# B&R Automation Studio project AP124 (part 2)

#### Variables.var - Local variables
```iecst
VAR
	closeArms : BOOL; (*VISU:1..command to close the arms, 0...open arms*)
	cmdDown : BOOL; (*VISU: button to go with magazine down*)
	cmdUp : BOOL; (*VISU: go with magazine down*)
	diActivateMagazineSafetyCircuits : BOOL; (*magazine:3 funkce v 1 (reset safety+ovladaci obvody + start automatu pokud jede paletizace)*)
	diLeftArmClosed : BOOL; (*left arm is closed*)
	diLeftArmOpened : BOOL; (*left arm is opened*)
	diMagazineLooseChain : BOOL; (*lower HW end switch*)
	diMagazineLowerPosition : BOOL; (*magazine in lower position*)
	diMagazineMiddlePositon : BOOL; (*magazine in middle position*)
	diMagazineUpperHwEnd : BOOL; (*upper HW end switch*)
	diMagazineUpperPosition : BOOL; (*magazine in upper position*)
	diMotorProtectionP11 : BOOL; (*contactor for vertical movement, 1=OK*)
	diPalletOnConveyorP12 : BOOL; (*pallet detected on conveyor P12*)
	diRightArmClosed : BOOL; (*right arm is closed*)
	diRightArmOpened : BOOL; (*right arm is opened*)
	doCloseArms : BOOL; (*valve to close the arms*)
	doLedP11 : BOOL;
	doMagazineBrake : BOOL; (*1=brake released*)
	doMagazineDown : BOOL; (*contactor to go down*)
	doMagazineUp : BOOL; (*contactor to go up*)
	doOpenArms : BOOL; (*valve to open the arms*)
	lightCurtainP11 : BOOL; (*status of light curtain P11*)
	MTBasicsPWM_0 : MTBasicsPWM;
	readyToStart : BOOL;
	stateArms : StateArms; (*VISU:arms state*)
	stateAuto : StateAuto;
	stateMagazine : StateMagazine; (*VISU: current state of magazine*)
	TON_LeftRequest : TON;
	TON_RightRequest : TON;
	TON_VerticalMovement : TON;
	TP_Start : TP;
	TON_PalletOnConveyorP12 : TON;
	modeZoneMagazineOld : ModeZone;
END_VAR
```

#### horizontalArmsControl.st
```iecst
(* control of arms *)

ACTION HorizontalArmsControl:

	IF modeZoneMagazine = modeZoneOff THEN
		stateArms := stateArmsInit;
	END_IF

	CASE stateArms OF

		stateArmsInit:

			IF diLeftArmClosed AND diRightArmClosed AND NOT diLeftArmOpened AND NOT diRightArmOpened THEN
				closeArms := TRUE;
				stateArms := stateArmsClosed;
			END_IF

			IF diLeftArmOpened AND diRightArmOpened AND NOT diLeftArmClosed AND NOT diRightArmClosed THEN
				closeArms := FALSE;
				stateArms := stateArmsOpened;
			END_IF

			//default state
			IF stateArms = stateArmsInit THEN
				doCloseArms := TRUE;
				doOpenArms := NOT doCloseArms;
			END_IF

		stateArmsOpening:

			//set output
			doCloseArms := FALSE;
			//invert second output
			doOpenArms := NOT doCloseArms;
			//start left timer
			TON_LeftRequest(IN := NOT diLeftArmOpened, PT := T#6s);
			//start right timer
			TON_RightRequest(IN := NOT diRightArmOpened, PT := T#6s);
			//open check
			IF diLeftArmOpened AND diRightArmOpened THEN
				stateArms := stateArmsOpened;
			END_IF
			//timeout left side?
			IF TON_LeftRequest.Q THEN
				alarmImageMagazine[4] := TRUE;
				closeArms := TRUE;
				stateArms := stateArmsClosed;
			END_IF
			//timeout right side?
			IF TON_RightRequest.Q THEN
				alarmImageMagazine[5] := TRUE;
				closeArms := TRUE;
				stateArms := stateArmsClosed;
			END_IF

		stateArmsOpened:

			// command to close
			IF closeArms THEN
				IF stateMagazine = stateUpperPosition THEN
					alarmImageMagazine[16] := TRUE;
					closeArms := FALSE;
				ELSE
					TON_LeftRequest(IN := FALSE);
					TON_RightRequest(IN := FALSE);
					stateArms := stateArmsClosing;
				END_IF
			END_IF

		stateArmsClosing:

			//set output
			doCloseArms := TRUE;
			//invert second output
			doOpenArms := NOT doCloseArms;
			//start left timer
			TON_LeftRequest(IN := NOT diLeftArmClosed, PT := T#6s);
			//start right timer
			TON_RightRequest(IN := NOT diRightArmClosed, PT := T#6s);
			//close check
			IF diLeftArmClosed AND diRightArmClosed THEN
				stateArms := stateArmsClosed;
			END_IF
			//timeout left side?
			IF TON_LeftRequest.Q THEN
				alarmImageMagazine[2] := TRUE;
				closeArms := FALSE;
				stateArms := stateArmsOpened;
			END_IF
			//timeout right side?
			IF TON_RightRequest.Q THEN
				alarmImageMagazine[3] := TRUE;
				closeArms := FALSE;
				stateArms := stateArmsOpened;
			END_IF

		stateArmsClosed:

			// command to open
			IF NOT closeArms THEN
				IF stateMagazine = stateLowerPosition OR (diReset AND stateMagazine <> stateUpperPosition) THEN
					TON_LeftRequest(IN := FALSE);
					TON_RightRequest(IN := FALSE);
					stateArms := stateArmsOpening;
				ELSE
					alarmImageMagazine[15] := TRUE;
					closeArms := TRUE;
				END_IF
			END_IF
	END_CASE

	//alarms
	IF stateArms = stateArmsInit THEN
		alarmImageMagazine[0] := TRUE;
	ELSE
		alarmImageMagazine[0] := FALSE;
	END_IF

	//edge alarms
	IF acknowledgeImageMagazine[2] THEN
		alarmImageMagazine[2] := FALSE;
	END_IF
	IF acknowledgeImageMagazine[3] THEN
		alarmImageMagazine[3] := FALSE;
	END_IF
	IF acknowledgeImageMagazine[4] THEN
		alarmImageMagazine[4] := FALSE;
	END_IF
	IF acknowledgeImageMagazine[5] THEN
		alarmImageMagazine[5] := FALSE;
	END_IF
	IF acknowledgeImageMagazine[15] THEN
		alarmImageMagazine[15] := FALSE;
	END_IF
	IF acknowledgeImageMagazine[16] THEN
		alarmImageMagazine[16] := FALSE;
	END_IF

END_ACTION
```

#### verticalArmsControl.st
```iecst
(* control of magazine *)

ACTION VerticalArmsControl:

	IF modeZoneMagazine = modeZoneOff THEN
		StopMovement;
	END_IF

	CASE stateMagazine OF
		stateMagazineUndefined:

			IF diMagazineUpperPosition AND NOT diMagazineMiddlePositon AND NOT diMagazineLowerPosition THEN
				stateMagazine := stateUpperPosition;
			END_IF

			IF NOT diMagazineUpperPosition AND diMagazineMiddlePositon AND NOT diMagazineLowerPosition THEN
				stateMagazine := stateMiddlePosition;
			END_IF

			IF NOT diMagazineUpperPosition AND NOT diMagazineMiddlePositon AND diMagazineLowerPosition THEN
				stateMagazine := stateLowerPosition;
			END_IF

			IF stateMagazine = stateMagazineUndefined THEN
				IF cmdDown THEN
					TON_VerticalMovement(IN := FALSE);
					stateMagazine := stateMoveToLowerPosition;
				END_IF

				IF cmdUp THEN
					TON_VerticalMovement(IN := FALSE);
					stateMagazine := stateMoveToUpperPosition;
				END_IF
			END_IF

		stateMoveToUpperPosition:
			//set output
			doMagazineUp := TRUE;
			//start timer
			TON_VerticalMovement(IN := TRUE, PT := T#6s);
			//position reached?
			IF diMagazineUpperPosition OR NOT cmdUp THEN
				StopMovement;
			END_IF
			//timeout?
			IF TON_VerticalMovement.Q THEN
				alarmImageMagazine[7] := TRUE;
				StopMovement;
			END_IF

		stateUpperPosition:

			IF cmdDown THEN
				IF statePalletP12 = palletPresent AND stateArms = stateArmsClosed THEN
					alarmImageMagazine[13] := TRUE;
					StopMovement;
				ELSE
					TON_VerticalMovement(IN := FALSE);
					stateMagazine := stateMoveToLowerPosition;
				END_IF
			END_IF
			cmdUp := FALSE;

		stateMoveLowerToMiddlePosition:
			//set output
			doMagazineUp := TRUE;
			//start timer
			TON_VerticalMovement(IN := TRUE, PT := T#6s);
			//position reached?
			IF diMagazineMiddlePositon OR NOT cmdUp THEN
				StopMovement;
			END_IF
			//timeout?
			IF TON_VerticalMovement.Q THEN
				alarmImageMagazine[8] := TRUE;
				StopMovement;
			END_IF

		stateMiddlePosition:

			IF cmdDown THEN
				IF statePalletP12 = palletPresent AND stateArms = stateArmsClosed THEN
					alarmImageMagazine[13] := TRUE;
					StopMovement;
				ELSE
					TON_VerticalMovement(IN := FALSE);
					stateMagazine := stateMoveToLowerPosition;
				END_IF
			END_IF

			IF cmdUp THEN
				TON_VerticalMovement(IN := FALSE);
				stateMagazine := stateMoveToUpperPosition;
			END_IF

		stateMoveToLowerPosition:
			//set output
			doMagazineDown := TRUE;
			//start timer
			TON_VerticalMovement(IN := TRUE, PT := T#6s);
			//position reached?
			IF diMagazineLowerPosition OR NOT cmdDown THEN
				StopMovement;
			END_IF
			//timeout?
			IF TON_VerticalMovement.Q THEN
				alarmImageMagazine[9] := TRUE;
				StopMovement;
			END_IF

		stateLowerPosition:

			IF cmdUp THEN
				TON_VerticalMovement(IN := FALSE);
				stateMagazine := stateMoveLowerToMiddlePosition;
			END_IF
			cmdDown := FALSE;

	END_CASE

	//brake control
	IF doMagazineUp OR doMagazineDown THEN
		doMagazineBrake := TRUE;
	ELSE
		doMagazineBrake := FALSE;
	END_IF

	IF diMagazineUpperHwEnd AND cmdUp THEN
		alarmImageMagazine[10] := TRUE;
	END_IF

	IF diMagazineLooseChain AND cmdDown THEN
		alarmImageMagazine[11] := TRUE;
	END_IF

	//edge alarms
	IF acknowledgeImageMagazine[7] THEN
		alarmImageMagazine[7] := FALSE;
	END_IF
	IF acknowledgeImageMagazine[8] THEN
		alarmImageMagazine[8] := FALSE;
	END_IF
	IF acknowledgeImageMagazine[9] THEN
		alarmImageMagazine[9] := FALSE;
	END_IF
	IF acknowledgeImageMagazine[10] THEN
		alarmImageMagazine[10] := FALSE;
	END_IF
	IF acknowledgeImageMagazine[11] THEN
		alarmImageMagazine[11] := FALSE;
	END_IF
	IF acknowledgeImageMagazine[13] THEN
		alarmImageMagazine[13] := FALSE;
	END_IF

END_ACTION

ACTION StopMovement:
	cmdUp := FALSE;
	cmdDown := FALSE;
	doMagazineDown := doMagazineUp :=  FALSE;
	stateMagazine := stateMagazineUndefined;
END_ACTION
```

#### conveyorP12Control.st
```iecst
ACTION ConveyorP12Control:

	//detect pallet on conveyor
	IF diPalletOnConveyorP12 AND (stateMagazine = stateUpperPosition OR stateArms = stateArmsOpened) THEN
		palletOnConveyorP12 := TRUE;
	END_IF

	IF modeMagazine = modeMagazineNotReadyToStart THEN
		stateConveyor := stateConveyorUndefined;
	END_IF

	CASE stateConveyor OF

		stateConveyorUndefined:
			stateConveyor := stateConveyorEmpty;

		//conveyor is empty
		stateConveyorEmpty:

			IF palletOnConveyorP12 THEN
				stateConveyor := stateConveyorOccupied;
			END_IF

		//conveyor is occupied
		stateConveyorOccupied:

			IF cmdMovePallet AND NOT palletOnConveyorP13 THEN
				TON_ConveyorP12(IN := FALSE);
				stateConveyor := stateConveyorMoving;
			END_IF

		//start conveyor
		stateConveyorMoving:
			doConveyorP12 := TRUE;
			//start timer
			TON_ConveyorP12(IN := TRUE, PT := T#6s);
			//sensor reached?
			IF palletOnConveyorP13 THEN
				palletOnConveyorP12 := FALSE;
				stateConveyor := stateConveyorStop;
			END_IF
			//timeout?
			IF TON_ConveyorP12.Q THEN
				alarmImage[14] := TRUE;
				stateConveyor := stateConveyorStop;
			END_IF

		//stop conveyor
		stateConveyorStop:
			doConveyorP12 := FALSE;
			stateConveyor := stateConveyorEmpty;

	END_CASE

	//edge alarms
	IF acknowledgeImage[14] THEN
		alarmImage[14] := FALSE;
	END_IF

END_ACTION
```

#### arms.st - not listed in the package file held
```iecst
(* control of arms *)

ACTION ArmsControl:

	CASE armsState OF
		stateArmsUndefined:

			IF diLeftArmClosed AND diRightArmClosed AND NOT diLeftArmOpened AND NOT diRightArmOpened THEN
				armsState := stateArmsClosed;
			END_IF

			IF diLeftArmOpened AND diRightArmOpened AND NOT diLeftArmClosed AND NOT diRightArmClosed THEN
				armsState := stateArmsOpened;
			END_IF

		stateArmsOpening:

			//set output
			doCloseArms := FALSE;
			//invert second output
			doOpenArms := NOT doCloseArms;
			//start left timer
			TON_LeftRequest(IN := NOT diLeftArmOpened, PT := T#6s);
			//start right timer
			TON_RightRequest(IN := NOT diRightArmOpened, PT := T#6s);
			//open check
			IF diLeftArmOpened AND diRightArmOpened THEN
				armsState := stateArmsOpened;
			END_IF
			//timeout left side?
			IF TON_LeftRequest.Q THEN
				MpAlarmXSet(gAlarmXCore,'LeftArmNotOpened');
				armsState := stateArmsClosed;
			END_IF
			//timeout right side?
			IF TON_RightRequest.Q THEN
				MpAlarmXSet(gAlarmXCore,'RightArmNotOpened');
				armsState := stateArmsClosed;
			END_IF

		stateArmsOpened:

			// command to close
			IF cmdCloseArms THEN
				TON_LeftRequest(IN := FALSE);
				TON_RightRequest(IN := FALSE);
				armsState := stateArmsClosing;
			END_IF

		stateArmsClosing:

			//set output
			doCloseArms := TRUE;
			//invert second output
			doOpenArms := NOT doCloseArms;
			//start left timer
			TON_LeftRequest(IN := NOT diLeftArmClosed, PT := T#6s);
			//start right timer
			TON_RightRequest(IN := NOT diRightArmClosed, PT := T#6s);
			//close check
			IF diLeftArmClosed AND diRightArmClosed THEN
				armsState := stateArmsClosed;
			END_IF
			//timeout left side?
			IF TON_LeftRequest.Q THEN
				MpAlarmXSet(gAlarmXCore,'LeftArmNotClosed');
				armsState := stateArmsOpened;
			END_IF
			//timeout right side?
			IF TON_RightRequest.Q THEN
				MpAlarmXSet(gAlarmXCore,'RightArmNotClosed');
				armsState := stateArmsOpened;
			END_IF

		stateArmsClosed:

			// command to open
			IF cmdOpenArms THEN
				TON_LeftRequest(IN := FALSE);
				TON_RightRequest(IN := FALSE);
				armsState := stateArmsOpening;
			END_IF

	END_CASE

END_ACTION
```

#### magazine.st - not listed in the package file held
```iecst
(* control of magazine *)

ACTION MagazineControl:

	CASE magazineState OF
		stateUndefined:

			IF diMagazineUpperPosition AND NOT diMagazineMiddlePositon AND NOT diMagazineLowerPosition THEN
				magazineState := stateUpperPosition;
			END_IF

			IF NOT diMagazineUpperPosition AND diMagazineMiddlePositon AND NOT diMagazineLowerPosition THEN
				magazineState := stateMiddlePosition;
			END_IF

			IF NOT diMagazineUpperPosition AND NOT diMagazineMiddlePositon AND diMagazineLowerPosition THEN
				magazineState := stateLowerPosition;
			END_IF

		stateMoveToUpperPosition:
			//set output
			doMagazineUp := TRUE;
			//start timer
			TON_VerticalMovement(IN := TRUE, PT := T#6s);
			//position reached?
			IF diMagazineUpperPosition THEN
				MagazineFinishMovement;
				magazineState := stateUpperPosition;
			END_IF
			//timeout?
			IF TON_VerticalMovement.Q THEN
				MagazineFinishMovement;
				MpAlarmXSet(gAlarmXCore,'UpperPositionNotReached');
				magazineState := stateMiddlePosition;
			END_IF

		stateUpperPosition:

			IF cmdDown THEN
				magazineState := stateMoveUpperToMiddlePosition;
			END_IF

		stateMoveUpperToMiddlePosition:

			//set output
			doMagazineDown := TRUE;
			//start timer
			TON_VerticalMovement(IN := TRUE, PT := T#6s);
			//position reached?
			IF diMagazineMiddlePositon THEN
				MagazineFinishMovement;
				magazineState := stateMiddlePosition;
			END_IF
			//timeout?
			IF TON_VerticalMovement.Q THEN
				MagazineFinishMovement;
				MpAlarmXSet(gAlarmXCore,'MiddlePositionNotReached');
				magazineState := stateUpperPosition;
			END_IF

		stateMoveLowerToMiddlePosition:
			//set output
			doMagazineUp := TRUE;
			//start timer
			TON_VerticalMovement(IN := TRUE, PT := T#6s);
			//position reached?
			IF diMagazineMiddlePositon THEN
				MagazineFinishMovement;
				magazineState := stateMiddlePosition;
			END_IF
			//timeout?
			IF TON_VerticalMovement.Q THEN
				MagazineFinishMovement;
				MpAlarmXSet(gAlarmXCore,'MiddlePositionNotReached');
				magazineState := stateLowerPosition;
			END_IF

		stateMiddlePosition:

			IF cmdDown THEN
				magazineState := stateMoveToLowerPosition;
			END_IF

			IF cmdUp THEN
				magazineState := stateMoveToUpperPosition;
			END_IF

		stateMoveToLowerPosition:
			//set output
			doMagazineDown := TRUE;
			//start timer
			TON_VerticalMovement(IN := TRUE, PT := T#6s);
			//position reached?
			IF diMagazineLowerPosition THEN
				MagazineFinishMovement;
				magazineState := stateLowerPosition;
			END_IF
			//timeout?
			IF TON_VerticalMovement.Q THEN
				MagazineFinishMovement;
				MpAlarmXSet(gAlarmXCore,'LowerPositionNotReached');
				magazineState := stateMiddlePosition;
			END_IF

		stateLowerPosition:
			IF cmdUp THEN
				magazineState := stateMoveLowerToMiddlePosition;
			END_IF

	END_CASE

	//brake control
	IF doMagazineUp OR doMagazineDown THEN
		doMagazineBrake := TRUE;
	ELSE
		doMagazineBrake := FALSE;
	END_IF

END_ACTION

ACTION MagazineFinishMovement:
	cmdUp := FALSE;
	cmdDown := FALSE;
	TON_VerticalMovement(IN := FALSE);
	doMagazineDown := doMagazineUp :=  FALSE;
END_ACTION
```

### palletization.typ
```iecst
TYPE
	RobotData : 	STRUCT
		layer : INT;
		placeFirstHalf : BOOL;
		placeSeparator : BOOL;
		placeSeparatorAbove : BOOL;
	END_STRUCT;
	PusherDrive : 	STRUCT
		cmdAbsolute : BOOL;
		cmdJogPlus : BOOL;
		cmdJogMinus : BOOL;
		tolerance : DINT;
		positions : ARRAY[0..5]OF DINT;
		speed : DINT;
		requestedPositionIndex : INT;
		actualPositionIndex : INT;
		actualPosition : DINT;
	END_STRUCT;
	StatePallet :
		(
		palletNotPresent,
		palletPresent,
		palletMoving
		);
	StateRobotAuto :
		(
		stateRobotAutoInit,
		stateRobotAutoGoHome,
		stateRobotAutoGoHome2,
		stateRobotAutoPrepareHead,
		stateRobotAutoPreGoToTable,
		stateRobotAutoGoingToTable,
		stateRobotAutoGoToTable,
		stateRobotAutoWaitForBottles,
		stateRobotAutoRailingDown,
		stateRobotAutoCenteringForward,
		stateRobotAutoSwitch1,
		stateRobotAutoSeparator,
		stateRobotAutoSeparator2,
		stateRobotAutoSeparator3,
		stateRobotAutoSeparator4,
		stateRobotAutoSeparator5,
		stateRobotAutoSeparator6,
		stateRobotAutoHideSuckers,
		stateRobotAutoHideSuckers2,
		stateRobotAutoWaitForPallet,
		stateRobotAutoPlaceFirstHalf,
		stateRobotAutoPlaceFirstHalf2,
		stateRobotAutoPlaceFirstHalf3,
		stateRobotAutoPlaceFirstHalf4,
		stateRobotAutoPlaceSecondHalf,
		stateRobotAutoPlaceSecondHalf2,
		stateRobotAutoPlaceSecondHalf3,
		stateRobotAutoPlaceSecondHalf4,
		stateRobotAutoPlaceSecondHalf5,
		stateRobotAutoPlaceSecondHalf6,
		stateRobotAutoSeparatorAbove
		);
	StateInterlayerAuto :
		(
		stateInterlayerAutoInit,
		stateInterlayerAutoGoDown,
		stateInterlayerAutoFill,
		stateInterlayerAutoEmpty
		);
	StateRoller :
		(
		stateRollerInit,
		stateRollerOpening,
		stateRollerOpened,
		stateRollerClosing,
		stateRollerClosed
		);
	StateCentering :
		(
		stateCenteringInit,
		stateCenteringMovingForward,
		stateCenteringForward,
		stateCenteringMovingBack,
		stateCenteringBack
		);
	StateRailing :
		(
		stateRailingInit,
		stateRailingMovingUp,
		stateRailingUp,
		stateRailingMovingDown,
		stateRailingDown
		);
	StateSuckers :
		(
		stateSuckersInit,
		stateSuckersMovingForward,
		stateSuckersForward,
		stateSuckersMovingBack,
		stateSuckersBack
		);
END_TYPE
```

### palletization.var
```iecst
VAR
	acknowledgeImagePalletization : ARRAY[0..39] OF BOOL;
	alarmImagePalletization : ARRAY[0..39] OF BOOL;
	alarmInZonePalletization : BOOL;
	cmdPalletizationAuto : BOOL; (*VISU:switches pallet magazine to automatic mode*)
	cmdPalletizationManual : BOOL;
	counterTraysBehindRotation : INT;
	counterTraysInRobotHead : INT;
	counterTraysOnTable : INT;
	modePalletization : ModePalletization;
	modePalletizationOld : ModePalletization;
END_VAR
VAR RETAIN
	nbOfLayersOnPallet : INT;
	nbOfTraysInHalfLayer : INT;
	nbOfTraysInRobotHead : INT;
	nbOfTraysOnP2 : INT;
	nbOfTraysOnTable : INT;
END_VAR
VAR
	pusherDrive : PusherDrive;
	statePalletP12 : StatePallet;
	statePalletP13 : StatePallet;
	statePalletP14 : StatePallet;
	statePalletP15 : StatePallet;
	statePalletP16 : StatePallet;
	statePalletP17 : StatePallet;
	PalletStatus_old : ARRAY[12..22] OF DINT;
	PalletStatus : ARRAY[12..22] OF DINT;
END_VAR
```

### Program Logical/plc/palletization/palletization_main (IEC) - palletization state machine

#### palletization_main.st - Init, cyclic, exit code
```iecst
PROGRAM _INIT

END_PROGRAM

PROGRAM _CYCLIC

	modeZonePalletizationOld := modeZonePalletization;

	readyToStart := NOT diPalletizationEDM;

	IF cpuIsSimulated THEN
		readyToStart := TRUE;
	END_IF

	IF NOT readyToStart THEN
		modeZonePalletization := modeZoneOff;
	END_IF

	CASE modeZonePalletization OF

		modeZoneOff: //the automat is not ready to start

			cmdPalletizationManual := FALSE;
			cmdPalletizationAuto := FALSE;

			IF readyToStart THEN
				modeZonePalletization := modeZoneManual;
			END_IF

		modeZoneManual:

			cmdPalletizationManual := FALSE;

			IF (NOT alarmInZonePalletization OR cpuIsSimulated)  AND cmdPalletizationAuto THEN
				modeZonePalletization := modeZoneAuto;
			END_IF

		modeZoneAuto:

			cmdPalletizationAuto := FALSE;

			IF (alarmInZonePalletization AND NOT cpuIsSimulated) OR cmdPalletizationManual THEN
				modeZonePalletization := modeZoneManual;
			END_IF

	END_CASE

	//alarms

END_PROGRAM
```

#### palletization_main.var - Local variables
```iecst
VAR
	readyToStart : BOOL;
	i : INT;
END_VAR
```

### Program Logical/plc/palletization/product_infeed/product_infeed (IEC) - product infeed control

#### Main.st - Cyclic code
```iecst
PROGRAM _INIT

	dNextTray ACCESS ADR(nullTray);
	dTrayBehindRotation ACCESS ADR(nullTray);

END_PROGRAM

PROGRAM _CYCLIC

	HMIS;
	RFRD;

	IF adrRecipes = 0 THEN
		RETURN;
	END_IF

	dRecipes ACCESS adrRecipes;
	IF dRecipes.actualRecipeIndex < 0 OR dRecipes.actualRecipeIndex > 9 THEN
		RETURN;
	END_IF

	dActualRecipe ACCESS ADR(dRecipes.recipe[dRecipes.actualRecipeIndex]);

	//correct wrong value in recipe
	IF dActualRecipe.nbOfLayers < 1 THEN
		dActualRecipe.nbOfLayers := 1;
	END_IF

	//select actual layout
	IF actualLayerIndex < 0 OR actualLayerIndex > 9 THEN
		RETURN;
	END_IF

	dActualLayout ACCESS ADR(dRecipes.layout[dActualRecipe.layer[actualLayerIndex]]);

	//the last tray in layout has to have set flag lastTrayInLayer
	dActualLayout.tray[dActualLayout.nbOfTrays - 1].lastTray := lastTrayInLayer;

	nbOfTraysInCompletePallet := dActualRecipe.nbOfLayers*dActualLayout.nbOfTrays;

	TOF_TrayOnOutputP1(IN := diTrayOnOutputP1, PT := T#10ms);
	TOF_TrayBehindRotation(IN := diTrayBehindRotation, PT := T#30ms);

	CASE modeZonePalletization OF

		modeZoneOff:

		modeZoneManual:

			IF modeZonePalletizationOld <> modeZoneManual THEN
				cmdRunConveyorP1 := FALSE;
				cmdRunConveyorP2 := FALSE;
				rotationForward := FALSE;
				bumperAuto := FALSE;
			END_IF

			acpI_P10.speed := 1000;
			acpI_P11.speed := 1200;
			pusherDrive.speed := 300;

			IF EDGEPOS(cmdRunConveyorsP1P2) THEN
				cmdRunConveyorP1 := TRUE;
				cmdRunConveyorP2 := TRUE;
			END_IF

			IF EDGENEG(cmdRunConveyorsP1P2) THEN
				cmdRunConveyorP1 := FALSE;
				cmdRunConveyorP2 := FALSE;
			END_IF

			automatMode := automatModeInit;

		modeZoneAuto:

			CASE automatMode OF
				automatModeInit:

					//initialize counters when program changes
					IF dRecipes.actualRecipeIndex <> actualRecipeIndexOld THEN
						nbOfLayersOnPallet := 0;
						nbOfTraysInHalfLayer := 0;
						nbOfTraysInRobotHead := 0;
						nbOfTraysOnTable := 0;
						nbOfTraysOnP2 := 0;
					END_IF
					actualRecipeIndexOld := dRecipes.actualRecipeIndex;

					counterTraysOnPallet := nbOfLayersOnPallet * dActualLayout.nbOfTrays;
					counterTraysOnPallet := counterTraysOnPallet + nbOfTraysInHalfLayer;
					counterTraysInRobotHead := (counterTraysOnPallet + nbOfTraysInRobotHead)(* MOD nbOfTraysInCompletePallet*);
					counterTraysOnTable := (counterTraysInRobotHead + nbOfTraysOnTable) (*MOD nbOfTraysInCompletePallet*);
					counterTraysBehindRotation := (counterTraysOnTable + nbOfTraysOnP2) (*MOD nbOfTraysInCompletePallet*);

					counterTraysOnConveyorP2 := counterTraysBehindRotation;

					IF dActualLayout.nbOfTrays > 0 THEN
						IF counterTraysBehindRotation > 0 THEN
							actualLayerIndex := (counterTraysBehindRotation - 1) / dActualLayout.nbOfTrays;
						ELSE
							actualLayerIndex := 0;
						END_IF
					END_IF

					IF counterTraysOnPallet  = nbOfTraysInCompletePallet THEN
						palletComplete := TRUE;
					END_IF

					TON_Parking(IN := FALSE);
					automatMode := automatModeParking;

				automatModeParking:

					cmdRunConveyorP2 := TRUE;

					TON_Parking(IN := TRUE, PT := T#5s);
					IF TON_Parking.Q THEN
						dTrayBehindRotation ACCESS ADR(dActualLayout.tray[(counterTraysBehindRotation - 1) MOD dActualLayout.nbOfTrays]);
						cmdRunConveyorP1 := dTrayBehindRotation.lastTray = lastTrayNo OR counterTraysBehindRotation = counterTraysOnTable;
						automatMode := automatModeRun;
					END_IF

				automatModeRun:

					//detect tray on output of conveyor P1
					IF TOF_TrayOnOutputP1.Q < trayOnOutputP1old THEN
						counterTraysOnConveyorP2 := counterTraysOnConveyorP2 MOD nbOfTraysInCompletePallet;
						counterTraysOnConveyorP2 := counterTraysOnConveyorP2 + 1;
						//reset timer
						TON_TransitTime(IN := FALSE);
					END_IF

					//select next tray
					dNextTray ACCESS ADR(dActualLayout.tray[counterTraysOnConveyorP2 MOD dActualLayout.nbOfTrays]);

					//detect tray behind rotation
					IF TOF_TrayBehindRotation.Q < trayBehindRotationOld THEN
						counterTraysBehindRotation := counterTraysBehindRotation MOD nbOfTraysInCompletePallet;
						counterTraysBehindRotation := counterTraysBehindRotation + 1;
					END_IF

					//select tray behind rotation
					IF counterTraysBehindRotation > 0 THEN
						dTrayBehindRotation ACCESS ADR(dActualLayout.tray[(counterTraysBehindRotation-1) MOD dActualLayout.nbOfTrays]);
					END_IF

					IF counterTraysBehindRotation = counterTraysOnTable THEN
						dTrayBehindRotation ACCESS ADR(nullTray);
					END_IF

					acpI_P10.speed := dActualRecipe.conveyorP1speed;
					acpI_P11.speed := dActualRecipe.conveyorP2speed;
					pusherDrive.speed := 500;
					bumperAuto := TRUE;

					CASE stateAuto OF

						stateAutoInit:

							stateAuto := stateAutoPusherToBasic;

						stateAutoPusherToBasic:

							pusherDrive.requestedPositionIndex := 1;
							pusherDrive.cmdAbsolute := TRUE;

							IF pusherDrive.actualPositionIndex = 1 THEN
								stateAuto := stateAutoPusherLiftingDown;
							END_IF

						stateAutoPusherLiftingDown:

							cmdPusherLiftingDown := TRUE;

							IF statePusherLifting = stateLowerPosition OR cpuIsSimulated THEN
								stateAuto := stateAutoFillRow;
							END_IF

						stateAutoFillRow:

							IF dTrayBehindRotation.lastTray <> lastTrayNo THEN
								stateAuto := stateAutoLastTray;
							END_IF

						stateAutoLastTray:

							TON_WaitForLastTray(IN := TRUE, PT := dActualRecipe.timeAfterLastTrayInRow);
							IF TON_WaitForLastTray.Q THEN
								cmdRunConveyorP1 := FALSE;
								IF dTrayBehindRotation.lastTray = lastTrayInRow THEN
									stateAuto := stateAutoPusherToTable;
								END_IF
								IF dTrayBehindRotation.lastTray = lastTrayInHalfLayer OR dTrayBehindRotation.lastTray = lastTrayInLayer THEN
									stateAuto := stateAutoPusherToRobotHead;
								END_IF
							END_IF

						stateAutoPusherToTable:

							IF diPusherBlockedByTray THEN
								alarmImagePalletization[28] := TRUE;
							ELSE
								stateAuto := stateAutoPusherToTable2;
							END_IF

						stateAutoPusherToTable2:

							pusherDrive.requestedPositionIndex := 2;
							pusherDrive.cmdAbsolute := TRUE;

							IF pusherDrive.actualPositionIndex = 2 THEN
								cmdRunConveyorP1 := TRUE;
								counterTraysOnTable := counterTraysBehindRotation;
								stateAuto := stateAutoPusherToBasic;
							END_IF

						stateAutoPusherLiftingUp:

							cmdPusherLiftingUp := TRUE;

							IF statePusherLifting = stateUpperPosition OR cpuIsSimulated THEN
								stateAuto := stateAutoPusherToBasic;
							END_IF

						stateAutoPusherToRobotHead:

							//wait for robot
							IF stateRobotAuto = stateRobotAutoWaitForBottles THEN
								IF stateRailing = stateRailingUp AND stateCentering = stateCenteringBack AND stateRoller = stateRollerClosed AND NOT diHeadIsFull AND nbOfTraysInRobotHead = 0 THEN
									stateAuto := stateAutoPusherToRobotHead2;
								END_IF
							END_IF

						stateAutoPusherToRobotHead2:

							//prepare data for robot
							robotData.layer := actualLayerIndex;
							robotData.placeFirstHalf := dTrayBehindRotation.lastTray = lastTrayInHalfLayer;

							IF actualLayerIndex = 0 THEN
								robotData.placeSeparator := dActualRecipe.interlayerSheetBottom;
							ELSE
								robotData.placeSeparator := TRUE;
							END_IF

							IF NOT robotData.placeFirstHalf THEN
								robotData.placeSeparator := FALSE;
							END_IF

							IF actualLayerIndex = dActualRecipe.nbOfLayers - 1 THEN
								robotData.placeSeparatorAbove := dActualRecipe.interlayerSheetTop;
							ELSE
								robotData.placeSeparatorAbove := FALSE;
							END_IF

							IF robotData.placeFirstHalf THEN
								robotData.placeSeparatorAbove := FALSE;
							END_IF

							//remember value for next states
							counterTraysOnTable := counterTraysBehindRotation;

							//correct counters
							IF dTrayBehindRotation.lastTray = lastTrayInLayer THEN
								//start new layer
								actualLayerIndex := actualLayerIndex + 1;
								IF actualLayerIndex = dActualRecipe.nbOfLayers THEN
									//new pallet, reset counters
//									counterTraysOnTable := 0;
									counterTraysBehindRotation := 0;
									counterTraysOnConveyorP2 := 0;
									actualLayerIndex := 0;
								END_IF
							END_IF

							stateAuto := stateAutoPusherToRobotHead3;

							dTrayBehindRotation ACCESS ADR(nullTray);

							//run conveyors
							cmdRunConveyorP1 := TRUE;

						stateAutoPusherToRobotHead3:

							//push to robot head
							IF diPusherBlockedByTray THEN
								alarmImagePalletization[28] := TRUE;
							ELSE
								stateAuto := stateAutoPusherToRobotHead4;
							END_IF

						stateAutoPusherToRobotHead4:

							pusherDrive.requestedPositionIndex := 4;
							pusherDrive.cmdAbsolute := TRUE;

							IF pusherDrive.actualPositionIndex = 4 THEN
								stateAuto := stateAutoPusherToRobotHead5;
							END_IF

						stateAutoPusherToRobotHead5:

							pusherDrive.requestedPositionIndex := 3;
							pusherDrive.cmdAbsolute := TRUE;

							IF pusherDrive.actualPositionIndex = 3 THEN
								//send data to robot
								counterTraysInRobotHead := counterTraysOnTable;
								IF counterTraysOnTable > counterTraysBehindRotation THEN
									counterTraysOnTable := 0;
								END_IF

//								robotData.start := TRUE;
								stateAuto := stateAutoPusherLiftingUp;
							END_IF
					END_CASE

					//control rotation only when no tray is in rotation zone
					IF counterTraysBehindRotation = counterTraysOnConveyorP2 THEN
						rotationForward := dNextTray.turnTray;
					END_IF

					//check sensor error
					TON_TransitTime(IN := TRUE, PT:=T#4s);
					IF TON_TransitTime.Q THEN
						IF counterTraysOnConveyorP2 > counterTraysBehindRotation THEN
							alarmImagePalletization[27] := TRUE;
						END_IF
						IF counterTraysOnConveyorP2 < counterTraysBehindRotation THEN
							alarmImagePalletization[55] := TRUE;
						END_IF
					END_IF

					//for start dialog
					nbOfLayersOnPallet := counterTraysOnPallet / dActualLayout.nbOfTrays;
					nbOfTraysInHalfLayer := counterTraysOnPallet MOD dActualLayout.nbOfTrays;
					nbOfTraysInRobotHead := (counterTraysInRobotHead - counterTraysOnPallet + nbOfTraysInCompletePallet) MOD nbOfTraysInCompletePallet;
					nbOfTraysOnTable := (counterTraysOnTable - counterTraysInRobotHead + nbOfTraysInCompletePallet) MOD nbOfTraysInCompletePallet;
					nbOfTraysOnP2 := (counterTraysBehindRotation - counterTraysOnTable + nbOfTraysInCompletePallet) MOD nbOfTraysInCompletePallet;

			END_CASE
	END_CASE

	trayOnOutputP1old := TOF_TrayOnOutputP1.Q;
	trayBehindRotationOld := TOF_TrayBehindRotation.Q;

	IF TON_WaitForLastTray.Q THEN
		TON_WaitForLastTray(IN := FALSE);
	END_IF

	ConveyorP1;
	ConveyorP2;
	PusherLifting;
	Rotation;
	Bumper;
	Interlayer;

	//door logic
	DoorLogic_1();
	alarmImagePalletization[39] := NOT DoorLogic_1.diDoorLocked;

	//edge alarms
	IF acknowledgeImagePalletization[27] THEN
		alarmImagePalletization[27] := FALSE;
	END_IF
	IF acknowledgeImagePalletization[28] THEN
		alarmImagePalletization[28] := FALSE;
	END_IF
	IF acknowledgeImagePalletization[55] THEN
		alarmImagePalletization[55] := FALSE;
	END_IF

	//problems with motors
	alarmImagePalletization[18] := NOT diMotorProtectionP3;

	alarmImagePalletization[22] := acpI_P10.error;
	acpI_P10.reset := EDGENEG(acknowledgeImagePalletization[22]);

	alarmImagePalletization[23] := acpI_P11.error;
	acpI_P11.reset := EDGENEG(acknowledgeImagePalletization[23]);

END_PROGRAM
```

#### Types.typ - Local data types
```iecst
TYPE
	AutomatMode :
		(
		automatModeInit,
		automatModeParking,
		automatModeRun
		);
	StateAuto :
		(
		stateAutoInit,
		stateAutoPusherToBasic,
		stateAutoPusherLiftingDown,
		stateAutoFillRow,
		stateAutoLastTray,
		stateAutoPusherToTable,
		stateAutoPusherToTable2,
		stateAutoPusherLiftingUp,
		stateAutoPusherToRobotHead,
		stateAutoPusherToRobotHead2,
		stateAutoPusherToRobotHead3,
		stateAutoPusherToRobotHead4,
		stateAutoPusherToRobotHead5
		);
	StateBumper :
		(
		stateBumperUndefined,
		stateBumperMovingForward,
		stateBumperForward,
		stateBumperMovingBack,
		stateBumperBack
		);
	StateConveyor :
		(
		stateConveyorStop,
		stateConveyorWait,
		stateConveyorMoving,
		stateConveyorPause,
		stateConveyorWaitForRotation,
		stateConveyorMoveTrayFromP1toP2,
		stateConveyorDelayForTurn,
		stateConveyorFillP1
		);
	StatePusherLifting :
		(
		statePusherLiftingUndefined,
		stateMoveToUpperPosition,
		stateUpperPosition,
		stateMoveToLowerPosition,
		stateLowerPosition
		);
	StateRotation :
		(
		stateRotationUndefined,
		stateRotationMovingForward,
		stateRotationForward,
		stateRotationMovingBack,
		stateRotationBack
		);
	StateInterlayer :
		(
		stateInterlayerInit,
		stateInterlayerDown,
		stateInterlayerGoUp,
		stateInterlayerUp,
		stateInterlayerGoDown,
		stateInterlayerGoDown2
		);
END_TYPE
```

#### Variables.var - Local variables
```iecst
VAR
	acpI_P10 : AcpInoSdc;
	acpI_P11 : AcpInoSdc;
	actualLayerIndex : INT;
END_VAR
VAR RETAIN
	actualRecipeIndexOld : INT;
END_VAR
VAR
	automatMode : AutomatMode;
	bumperAuto : BOOL;
	bumperForward : BOOL;
	cmdInterlayerDown : BOOL;
	cmdInterlayerUp : BOOL;
	cmdPusherLiftingDown : BOOL;
	cmdPusherLiftingUp : BOOL;
	cmdRunConveyorP1 : BOOL;
	cmdRunConveyorP2 : BOOL;
	cmdRunConveyorsP1P2 : BOOL;
	counterTraysOnConveyorP2 : INT;
	dActualLayout : REFERENCE TO Layout;
	dActualRecipe : REFERENCE TO Recipe;
	diBumperForward : BOOL;
	diInterlayerDown : BOOL;
	diInterlayerSafeFrame : BOOL;
	diInterlayerUp : BOOL;
	diInterlayerUpperHwEnd : BOOL;
	diMotorProtectionP3 : BOOL;
	diNoInterlayerSheet : BOOL;
	diPusherBlockedByTray : BOOL;
	diPusherLiftingLowerPosition : BOOL;
	diPusherLiftingUpperPosition : BOOL;
	diRotationBack : BOOL;
	diRotationForward : BOOL;
	diTrayBehindRotation : BOOL;
	diTrayOnInputP1 : BOOL;
	diTrayOnOutputP1 : BOOL;
	dNextTray : REFERENCE TO Tray;
	doBumper : BOOL;
	doInterlayerDown : BOOL;
	doInterlayerEnable : BOOL;
	doInterlayerPowerOn : BOOL;
	doInterlayerUp : BOOL;
	DoorLogic_1 : DoorLogic;
	doPusherLiftingBrake : BOOL;
	doPusherLiftingDown : BOOL;
	doPusherLiftingUp : BOOL;
	doRotationBack : BOOL;
	doRotationForward : BOOL;
	dRecipes : REFERENCE TO Recipes;
	dTrayBehindRotation : REFERENCE TO Tray;
	HMIS : UINT;
	nullTray : Tray;
	RFRD : INT;
	rotationForward : BOOL; (*1..requested forward,0..requested back*)
	stateAuto : StateAuto;
	stateBumper : StateBumper;
	stateConveyorP1 : StateConveyor;
	stateConveyorP2 : StateConveyor;
	stateInterlayer : StateInterlayer;
	statePusherLifting : StatePusherLifting;
	stateRotation : StateRotation;
	TOF_TrayBehindRotation : TOF;
	TOF_TrayOnInputP1 : TOF;
	TOF_TrayOnOutputP1 : TOF;
	TON_Bumper : TON;
	TON_JumpUp : TON;
	TON_Parking : TON;
	TON_RotationRequest : TON;
	TON_TransitTime : TON;
	TON_TurnTray : TON;
	TON_VerticalMovement : TON;
	TON_WaitForLastTray : TON;
	trayBehindRotationOld : BOOL;
	trayOnOutputP1old : BOOL;
	TOF_acpI_P10 : TOF;
END_VAR
```

#### conveyorP1.st
```iecst
ACTION ConveyorP1:

	IF modeZonePalletization = modeZoneOff OR (modeZonePalletizationOld = modeZoneAuto AND modeZonePalletization <> modeZoneAuto) THEN
		stateConveyorP1 := stateConveyorStop;
	END_IF

	//pause conveyor when no trays on input
	TOF_TrayOnInputP1(IN := diTrayOnInputP1 OR diTrayOnOutputP1, PT := T#10s);

	CASE stateConveyorP1 OF

		stateConveyorStop:

			//cmdRunConveyorP1 := FALSE;
			acpI_P10.switchOn := TRUE;
			acpI_P10.run := FALSE;
			IF modeZonePalletization <> modeZoneOff THEN
				stateConveyorP1 := stateConveyorWait;
			END_IF

		stateConveyorWait:

			IF cmdRunConveyorP1 THEN
				TOF_TrayOnInputP1(IN:=TRUE);
				stateConveyorP1 := stateConveyorMoving;
			END_IF

		stateConveyorMoving:

			acpI_P10.run := TRUE;

			IF modeZonePalletization = modeZoneAuto THEN
				//pause?
				IF NOT TOF_TrayOnInputP1.Q THEN
					stateConveyorP1 := stateConveyorPause;
				END_IF

				//detection of new tray
				IF TOF_TrayOnOutputP1.Q THEN
					stateConveyorP1 := stateConveyorWaitForRotation;
				END_IF
			END_IF

			IF NOT cmdRunConveyorP1 THEN
				stateConveyorP1 := stateConveyorStop;
			END_IF

		stateConveyorPause:

			acpI_P10.run := FALSE;

			//wake up
			IF TOF_TrayOnInputP1.Q THEN
				stateConveyorP1 := stateConveyorMoving;
			END_IF

		stateConveyorWaitForRotation:

			//stop request?
			IF dNextTray.lastTray <> lastTrayNo THEN
				cmdRunConveyorP1 := FALSE;
			END_IF

			//wait till rotation is in correct place
			acpI_P10.run := FALSE;

			IF dNextTray.turnTray THEN
				IF stateRotation = stateRotationForward THEN
					stateConveyorP1 := stateConveyorMoveTrayFromP1toP2;
				END_IF
			ELSE
				IF stateRotation = stateRotationBack THEN
					stateConveyorP1 := stateConveyorMoveTrayFromP1toP2;
				END_IF
			END_IF

		stateConveyorMoveTrayFromP1toP2:

			//move tray from P1 to P2
			acpI_P10.run := TRUE;

			IF NOT TOF_TrayOnOutputP1.Q THEN
				TON_TurnTray(IN:=FALSE);
				stateConveyorP1 := stateConveyorDelayForTurn;
			END_IF

		stateConveyorDelayForTurn:

			//time delay for turn
			acpI_P10.run := FALSE;

			TON_TurnTray(IN:=TRUE, PT := dActualRecipe.timeDelayForTurn);
			IF TON_TurnTray.Q OR stateRotation = stateRotationBack THEN
				stateConveyorP1 := stateConveyorFillP1;
			END_IF

		stateConveyorFillP1:

			//fill conveyor P1
			acpI_P10.run := TRUE;

			//pause?
			IF NOT TOF_TrayOnInputP1.Q THEN
				stateConveyorP1 := stateConveyorMoving;
			END_IF

			//tray detected
			IF TOF_TrayOnOutputP1.Q THEN
				stateConveyorP1 := stateConveyorMoving;
			END_IF

	END_CASE

	//control of ACOPOSinverter P14
	acpI_P10();

END_ACTION
```

#### conveyorP2.st
```iecst
ACTION ConveyorP2:

	TOF_acpI_P10(IN := acpI_P10.run OR pusherDrive.cmdAbsolute, PT := T#10s);

	IF modeZonePalletization = modeZoneOff OR (modeZonePalletizationOld = modeZoneAuto AND modeZonePalletization <> modeZoneAuto) THEN
		stateConveyorP2 := stateConveyorStop;
	END_IF

	CASE stateConveyorP2 OF

		stateConveyorStop:

			acpI_P11.switchOn := TRUE;
			acpI_P11.run := FALSE;
			IF modeZonePalletization <> modeZoneOff THEN
				stateConveyorP2 := stateConveyorWait;
			END_IF

		stateConveyorWait:

			IF cmdRunConveyorP2 THEN
				TOF_acpI_P10(IN := TRUE);
				stateConveyorP2 := stateConveyorMoving;
			END_IF

		stateConveyorMoving:

			acpI_P11.run := TRUE;

			IF modeZonePalletization = modeZoneAuto THEN
				//pause?
				IF NOT TOF_acpI_P10.Q THEN
					stateConveyorP2 := stateConveyorPause;
				END_IF

			END_IF

			IF NOT cmdRunConveyorP2 THEN
				stateConveyorP2 := stateConveyorStop;
			END_IF

		stateConveyorPause:

			acpI_P11.run := FALSE;

			//wake up
			IF TOF_acpI_P10.Q THEN
				stateConveyorP2 := stateConveyorMoving;
			END_IF

	END_CASE

	//control of ACOPOSinverter
	acpI_P11();

END_ACTION
```

#### PusherLifting.st
```iecst
(* control of magazine *)

ACTION PusherLifting:

	IF modeZonePalletization = modeZoneOff THEN
		StopMovement;
	END_IF

	CASE statePusherLifting OF
		statePusherLiftingUndefined:

			IF diPusherLiftingUpperPosition AND NOT diPusherLiftingLowerPosition THEN
				statePusherLifting := stateUpperPosition;
			END_IF

			IF NOT diPusherLiftingUpperPosition AND diPusherLiftingLowerPosition THEN
				statePusherLifting := stateLowerPosition;
			END_IF

			IF statePusherLifting = statePusherLiftingUndefined THEN
				IF cmdPusherLiftingDown THEN
					TON_VerticalMovement(IN := FALSE);
					statePusherLifting := stateMoveToLowerPosition;
				END_IF

				IF cmdPusherLiftingUp THEN
					TON_VerticalMovement(IN := FALSE);
					statePusherLifting := stateMoveToUpperPosition;
				END_IF
			END_IF

		stateMoveToUpperPosition:
			//set output
			doPusherLiftingUp := TRUE;
			//start timer
			TON_VerticalMovement(IN := TRUE, PT := T#3s);
			//position reached?
			IF diPusherLiftingUpperPosition OR NOT cmdPusherLiftingUp THEN
				StopMovement;
			END_IF
			//timeout?
			IF TON_VerticalMovement.Q THEN
				alarmImagePalletization[16] := TRUE;
				StopMovement;
			END_IF

		stateUpperPosition:

			IF cmdPusherLiftingDown THEN
				TON_VerticalMovement(IN := FALSE);
				statePusherLifting := stateMoveToLowerPosition;
			END_IF
			cmdPusherLiftingUp := FALSE;

		stateMoveToLowerPosition:
			//set output
			doPusherLiftingDown := TRUE;
			//start timer
			TON_VerticalMovement(IN := TRUE, PT := T#3s);
			//position reached?
			IF diPusherLiftingLowerPosition OR NOT cmdPusherLiftingDown THEN
				StopMovement;
			END_IF
			//timeout?
			IF TON_VerticalMovement.Q THEN
				alarmImagePalletization[17] := TRUE;
				StopMovement;
			END_IF

		stateLowerPosition:

			IF cmdPusherLiftingUp THEN
				TON_VerticalMovement(IN := FALSE);
				statePusherLifting := stateMoveToUpperPosition;
			END_IF
			cmdPusherLiftingDown := FALSE;

	END_CASE

	//brake control
	doPusherLiftingBrake := doPusherLiftingUp OR doPusherLiftingDown;

	//edge alarms
	IF acknowledgeImagePalletization[16] THEN
		alarmImagePalletization[16] := FALSE;
	END_IF
	IF acknowledgeImagePalletization[17] THEN
		alarmImagePalletization[17] := FALSE;
	END_IF
END_ACTION

ACTION StopMovement:
	cmdPusherLiftingUp := FALSE;
	cmdPusherLiftingDown := FALSE;
	doPusherLiftingDown := doPusherLiftingUp :=  FALSE;
	statePusherLifting := statePusherLiftingUndefined;
END_ACTION
```

#### Rotation.st
```iecst
ACTION Rotation:

	IF modeZonePalletization = modeZoneOff THEN
		stateRotation := stateRotationUndefined;
	END_IF

	CASE stateRotation OF

		stateRotationUndefined:

			IF diRotationBack AND NOT diRotationForward THEN
				rotationForward := FALSE;
				stateRotation := stateRotationBack;
			END_IF

			IF NOT diRotationBack AND diRotationForward THEN
				rotationForward := TRUE;
				stateRotation := stateRotationForward;
			END_IF

			IF stateRotation = stateRotationUndefined THEN
				//set output
				doRotationForward := FALSE;
				//invert second output
				doRotationBack := NOT doRotationForward;
			END_IF

		stateRotationMovingForward:

			//set output
			doRotationForward := TRUE;
			//invert second output
			doRotationBack := NOT doRotationForward;
			//check
			IF diRotationForward THEN
				stateRotation := stateRotationForward;
			END_IF
			// timer
			TON_RotationRequest(IN := NOT diRotationForward, PT := T#5s);
			IF TON_RotationRequest.Q THEN
				rotationForward := FALSE;
				alarmImagePalletization[20] := TRUE;
				stateRotation := stateRotationBack;
			END_IF

		stateRotationForward:

			// command back
			IF NOT rotationForward THEN
				TON_RotationRequest(IN := FALSE);
				stateRotation := stateRotationMovingBack;
			END_IF

		stateRotationMovingBack:

			//set output
			doRotationBack := TRUE;
			//invert second output
			doRotationForward := NOT doRotationBack;
			//check
			IF diRotationBack THEN
				stateRotation := stateRotationBack;
			END_IF
			// timer
			TON_RotationRequest(IN := NOT diRotationBack, PT := T#5s);
			IF TON_RotationRequest.Q THEN
				rotationForward := TRUE;
				alarmImagePalletization[21] := TRUE;
				stateRotation := stateRotationForward;
			END_IF

		stateRotationBack:

			// command forward
			IF rotationForward THEN
				TON_RotationRequest(IN := FALSE);
				stateRotation := stateRotationMovingForward;
			END_IF
	END_CASE

	//alarms
	IF stateRotation = stateRotationUndefined THEN
		alarmImagePalletization[19] := TRUE;
	ELSE
		alarmImagePalletization[19] := FALSE;
	END_IF

	//edge alarms
	IF acknowledgeImagePalletization[20] THEN
		alarmImagePalletization[20] := FALSE;
	END_IF
	IF acknowledgeImagePalletization[21] THEN
		alarmImagePalletization[21] := FALSE;
	END_IF

END_ACTION
```

#### Bumper.st
```iecst
ACTION Bumper:

	IF modeZonePalletization = modeZoneOff THEN
		stateBumper := stateBumperUndefined;
	END_IF

	CASE stateBumper OF

		stateBumperUndefined:

			IF diBumperForward THEN
				stateBumper := stateBumperForward;
			ELSE
				stateBumper := stateBumperBack;
			END_IF

		stateBumperMovingForward:

			doBumper := TRUE;

			IF diBumperForward THEN
				stateBumper := stateBumperForward;
			END_IF

		stateBumperForward:

			IF bumperAuto THEN
				bumperForward := FALSE;
			END_IF

			IF NOT bumperForward THEN
				stateBumper := stateBumperMovingBack;
			END_IF

		stateBumperMovingBack:

			doBumper := FALSE;

			IF NOT diBumperForward THEN
				TON_Bumper(IN:=FALSE);
				stateBumper := stateBumperBack;
			END_IF

		stateBumperBack:

			TON_Bumper(IN:=TRUE,PT:=T#0.2s);
			IF bumperAuto AND TON_Bumper.Q THEN
				bumperForward := TRUE;
			END_IF

			IF bumperForward THEN
				stateBumper := stateBumperMovingForward;
			END_IF

	END_CASE
END_ACTION
```

#### Interlayer.st
```iecst
ACTION Interlayer:

	doInterlayerEnable := modeZonePalletization <> modeZoneOff;
	doInterlayerPowerOn := TRUE;

//	diInterlayerSheetPresent;

	IF modeZonePalletization = modeZoneOff THEN
		stateInterlayer := stateInterlayerInit;
	END_IF

	CASE stateInterlayer OF

		stateInterlayerInit:

			IF diInterlayerUp AND NOT diInterlayerDown THEN
				stateInterlayer := stateInterlayerUp;
			END_IF

			IF NOT diInterlayerUp AND diInterlayerDown THEN
				stateInterlayer := stateInterlayerDown;
			END_IF

			IF stateInterlayer = stateInterlayerInit THEN
				IF cmdInterlayerUp THEN
					stateInterlayer := stateInterlayerGoUp;
				END_IF

				IF cmdInterlayerDown THEN
					stateInterlayer := stateInterlayerGoDown;
				END_IF
			END_IF

		stateInterlayerGoUp:

			//set output
			doInterlayerUp := TRUE;

			//position reached?
			IF diInterlayerUp OR NOT diNoInterlayerSheet OR NOT cmdInterlayerUp THEN
				StopInterlayer;
			END_IF

		stateInterlayerUp:

			IF cmdInterlayerDown THEN
				stateInterlayer := stateInterlayerGoDown;
			END_IF
			cmdInterlayerUp := FALSE;

		stateInterlayerGoDown:

			//first go up
			doInterlayerUp := TRUE;
			doInterlayerDown := FALSE;

			TON_JumpUp(IN := TRUE, PT := T#0.05s);
			IF TON_JumpUp.Q THEN
				stateInterlayer := stateInterlayerGoDown2;
			END_IF

		stateInterlayerGoDown2:

			//set output
			doInterlayerUp := FALSE;
			doInterlayerDown := TRUE;

			//position reached?
			IF diInterlayerDown OR NOT cmdInterlayerDown THEN
				StopInterlayer;
			END_IF

		stateInterlayerDown:

			IF cmdInterlayerUp THEN
				stateInterlayer := stateInterlayerGoUp;
			END_IF
			cmdInterlayerDown := FALSE;
	END_CASE

	CASE modeZonePalletization OF

		modeZoneOff:

		modeZoneManual:

			IF modeZonePalletizationOld <> modeZoneManual THEN
				cmdInterlayerUp := FALSE;
				cmdInterlayerDown := FALSE;
				interlayerSheetMagazineEmpty := FALSE;
			END_IF

			stateInterlayerAuto := stateInterlayerAutoInit;

		modeZoneAuto:

			CASE stateInterlayerAuto OF

				stateInterlayerAutoInit:

					stateInterlayerAuto := stateInterlayerAutoGoDown;

				stateInterlayerAutoGoDown:

					IF diNoInterlayerSheet THEN
						stateInterlayerAuto := stateInterlayerAutoFill;
					ELSE
						cmdInterlayerDown := TRUE;
					END_IF
					cmdInterlayerUp := FALSE;

				stateInterlayerAutoFill:

					IF diNoInterlayerSheet THEN
						cmdInterlayerUp := TRUE;
					END_IF
					cmdInterlayerDown := FALSE;

					IF stateInterlayer = stateInterlayerUp THEN
						stateInterlayerAuto := stateInterlayerAutoEmpty;
					END_IF

				stateInterlayerAutoEmpty:

					interlayerSheetMagazineEmpty := TRUE;
					cmdInterlayerDown := TRUE;

			END_CASE

	END_CASE

	alarmImagePalletization[43] := diInterlayerUpperHwEnd;
	alarmImagePalletization[44] := diInterlayerSafeFrame;

END_ACTION

ACTION StopInterlayer:
	cmdInterlayerUp := FALSE;
	cmdInterlayerDown := FALSE;
	doInterlayerUp := doInterlayerDown :=  FALSE;
	stateInterlayer := stateInterlayerInit;
	TON_JumpUp(IN := FALSE);
END_ACTION
```

#### PusherDriveP12.st - not listed in the package file held
```iecst
ACTION PusherDriveP12:

	IF modePalletization = modePalletizationNotReadyToStart THEN
		statePusherDriveP12 := statePusherDriveStop;
	END_IF

	CASE statePusherDriveP12 OF

		statePusherDriveStop:

			acpI_P12.switchOn := TRUE;
			acpI_P12.speed := 0;
			acpI_P12.reset := TRUE;

			FI_12.cmd.power := 1;

			IF modePalletization <> modePalletizationNotReadyToStart AND FI_12.info.powerOn THEN
				statePusherDriveP12 := statePusherDriveWait;
			END_IF

		statePusherDriveWait:

			IF NOT FI_12.info.homingOk THEN
				FI_12.param.position := 265;//homing position
				FI_12.param.speed := 50;
				FI_12.param.acceleration := 1000;
				FI_12.param.deceleration := 1000;
				FI_12.param.homing.mode := 2;
				FI_12.param.homing.startDirection := 1;
				FI_12.param.homing.edgeSwitch := 1;
				FI_12.param.homing.speed2 := 10;
				FI_12.cmd.homing := 1;
				statePusherDriveP12 := statePusherDriveHoming;
			END_IF

		statePusherDriveHoming:

			IF FI_12.info.homingOk THEN
				statePusherDriveP12 := statePusherDriveWait;
			END_IF

	END_CASE

	FI_12();
	acpI_P12();
	//acpI_P12.switchOn := FI_12.info.powerOn;

END_ACTION
```

### Program Logical/plc/palletization/product_infeed/pusher_drive (IEC) - pusher drive P12

#### Types.typ
```iecst
TYPE
	StatePusherDrive :
		(
		statePusherDriveUndefined,
		statePusherDriveStop,
		statePusherDriveHoming,
		statePusherDriveHoming2,
		statePusherDriveWait,
		statePusherDriveAbsolute,
		statePusherDriveAbsolute2,
		statePusherDriveJogPlus,
		statePusherDriveJogPlus2,
		statePusherDriveJogMinus,
		statePusherDriveJogMinus2
		);
END_TYPE
```

#### Variables.var
```iecst
VAR
	acpI_P12 : AcpInoSdc;
	FI_12 : FI;
	statePusherDriveP12 : StatePusherDrive;
	aoPusherDriveP12 : INT;
	oldMoveActive : BOOL;
	aiDistanceSensor : INT; (*SICK DL50*)
	actualPosition : DINT;
	i : INT;
END_VAR
```

#### Main.st
```iecst
PROGRAM _INIT
	FI_12.init.positiveSwLimit := 2300;
	FI_12.init.negativeSwLimit := 200;
	FI_12.init.taskTime := 0.01;
	FI_12.init.units := FI_12.init.positiveSwLimit-FI_12.init.negativeSwLimit;
	FI_12.init.encoderIncrements := 32537;
	FI_12.init.reverseDirection := 0;
	FI_12.init.maxLagError := 200;
	FI_12.init.Kp := 10;
	FI_12.init.Tn := 0;
	FI_12.init.speedFilter := 100;
	FI_12.init.settleTime := 0.5;

	pusherDrive.tolerance := 30;
	pusherDrive.positions[0] := FI_12.init.negativeSwLimit + pusherDrive.tolerance;
	pusherDrive.positions[1] := 925;
	pusherDrive.positions[2] := 1470;
	pusherDrive.positions[3] := 1650;
	pusherDrive.positions[4] := 1920;
	pusherDrive.positions[5] := 2000;//FI_12.init.positiveSwLimit-tolerance;
	pusherDrive.speed := 500;

	acpI_P12.run := TRUE;

END_PROGRAM

PROGRAM _CYCLIC

	actualPosition := FI_12.init.units*INT_TO_DINT(aiDistanceSensor)/32767+FI_12.init.negativeSwLimit;

	IF modeZonePalletization = modeZoneOff OR (modeZonePalletizationOld = modeZoneAuto AND modeZonePalletization <> modeZoneAuto) THEN
		statePusherDriveP12 := statePusherDriveStop;
	END_IF

	CASE statePusherDriveP12 OF

		statePusherDriveUndefined:

			FOR i := 0 TO 5 DO
				IF actualPosition >= pusherDrive.positions[i] - pusherDrive.tolerance AND  actualPosition <= pusherDrive.positions[i] + pusherDrive.tolerance THEN
					EXIT;
				END_IF
			END_FOR
			IF i <= 5 THEN
				pusherDrive.actualPositionIndex := i;
			ELSE
				pusherDrive.actualPositionIndex := 0;
			END_IF
			statePusherDriveP12 := statePusherDriveStop;

		statePusherDriveStop:

			acpI_P12.switchOn := FALSE;
			FI_12.cmd.power := FALSE;

			pusherDrive.cmdAbsolute := FALSE;
			pusherDrive.cmdJogPlus := FALSE;
			pusherDrive.cmdJogMinus := FALSE;

			IF modeZonePalletization <> modeZoneOff THEN
				statePusherDriveP12 := statePusherDriveWait;
			END_IF

		statePusherDriveWait:

			IF pusherDrive.cmdJogPlus THEN
				statePusherDriveP12 := statePusherDriveJogPlus;
			END_IF

			IF pusherDrive.cmdJogMinus THEN
				statePusherDriveP12 := statePusherDriveJogMinus;
			END_IF

			IF pusherDrive.cmdAbsolute THEN
				statePusherDriveP12 := statePusherDriveAbsolute;
			END_IF

			IF NOT FI_12.info.homingOk THEN
				statePusherDriveP12 := statePusherDriveHoming;
			END_IF

		statePusherDriveHoming:

			//compute actual position
			FI_12.param.position := actualPosition;
			FI_12.param.homing.mode := 0;
			FI_12.cmd.homing := 1;
			statePusherDriveP12 := statePusherDriveHoming2;

		statePusherDriveHoming2:

			IF FI_12.info.homingOk THEN
				statePusherDriveP12 := statePusherDriveStop;
			END_IF

		statePusherDriveAbsolute:

			FI_12.cmd.power := 1;
			acpI_P12.switchOn := TRUE;

			IF FI_12.info.powerOn AND acpI_P12.switchedOn THEN
				FI_12.cmd.absolute := TRUE;
				FI_12.param.position := pusherDrive.positions[pusherDrive.requestedPositionIndex];
				FI_12.param.speed := pusherDrive.speed;
				statePusherDriveP12 := statePusherDriveAbsolute2;
			END_IF

		statePusherDriveAbsolute2:

			IF NOT pusherDrive.cmdAbsolute THEN
				FI_12.cmd.stop := TRUE;
			END_IF

			IF oldMoveActive > FI_12.info.moveActive THEN
				pusherDrive.actualPositionIndex := pusherDrive.requestedPositionIndex;
				statePusherDriveP12 := statePusherDriveStop;
			END_IF

		statePusherDriveJogPlus:

			FI_12.cmd.power := 1;
			acpI_P12.switchOn := TRUE;

			IF FI_12.info.powerOn AND acpI_P12.switchedOn THEN

				pusherDrive.requestedPositionIndex := pusherDrive.actualPositionIndex + 1;
				IF pusherDrive.requestedPositionIndex > 5 THEN
					pusherDrive.requestedPositionIndex := 5;
				END_IF

				FI_12.cmd.absolute := TRUE;
				FI_12.param.position := pusherDrive.positions[pusherDrive.requestedPositionIndex];
				FI_12.param.speed := pusherDrive.speed;
				statePusherDriveP12 := statePusherDriveJogPlus2;
			END_IF

		statePusherDriveJogPlus2:

			IF NOT pusherDrive.cmdJogPlus THEN
				FI_12.cmd.stop := TRUE;
			END_IF

			//IF oldMoveActive > FI_12.info.moveActive THEN
			IF NOT FI_12.info.moveActive THEN
				pusherDrive.actualPositionIndex := pusherDrive.requestedPositionIndex;
				statePusherDriveP12 := statePusherDriveStop;
			END_IF

		statePusherDriveJogMinus:

			FI_12.cmd.power := 1;
			acpI_P12.switchOn := TRUE;

			IF FI_12.info.powerOn AND acpI_P12.switchedOn THEN
				pusherDrive.requestedPositionIndex := pusherDrive.actualPositionIndex - 1;
				IF pusherDrive.requestedPositionIndex < 1 THEN
					pusherDrive.requestedPositionIndex := 1;
				END_IF

				FI_12.cmd.absolute := TRUE;
				FI_12.param.position := pusherDrive.positions[pusherDrive.requestedPositionIndex];
				FI_12.param.speed := pusherDrive.speed;
				statePusherDriveP12 := statePusherDriveJogMinus2;
			END_IF

		statePusherDriveJogMinus2:

			IF NOT pusherDrive.cmdJogMinus THEN
				FI_12.cmd.stop := TRUE;
			END_IF

			IF NOT FI_12.info.moveActive THEN
				pusherDrive.actualPositionIndex := pusherDrive.requestedPositionIndex;
				statePusherDriveP12 := statePusherDriveStop;
			END_IF
	END_CASE

	oldMoveActive :=  FI_12.info.moveActive;

	memcpy(ADR(FI_12.IOMapping.Encoder), ADR(aiDistanceSensor), 2);
	FI_12();
	acpI_P12();

	aoPusherDriveP12 := FI_12.IOMapping.AnalogOutput;
	pusherDrive.actualPosition := FI_12.info.position;

	alarmImagePalletization[15] := aiDistanceSensor < -4000 OR aiDistanceSensor = 32767;

	alarmImagePalletization[14] := FI_12.info.status <> 0 OR acpI_P12.error;

	IF EDGENEG(acknowledgeImagePalletization[14]) THEN
		acpI_P12.reset := TRUE;
		FI_12.cmd.acknowledge := TRUE;
	END_IF

	IF cpuIsSimulated THEN
		pusherDrive.actualPositionIndex := pusherDrive.requestedPositionIndex;
	END_IF

END_PROGRAM
```

### Program Logical/plc/palletization/robot_head/robot_head (IEC) - robot head control

#### Main.st - Cyclic code
```iecst
PROGRAM _INIT

END_PROGRAM

PROGRAM _CYCLIC

	CASE modeZonePalletization OF

		modeZoneOff: //the automat is not ready to start

		modeZoneManual:

			IF modeZonePalletizationOld <> modeZoneManual THEN

			END_IF

		modeZoneAuto:

	END_CASE

	Railing;
	Suckers;
	Centering;
	Roller;

	//door logic
	DoorLogic_3();
	alarmImagePalletization[42] := NOT DoorLogic_3.diDoorLocked;

END_PROGRAM
```

#### Types.typ - Local data types
```iecst
TYPE
	StateRoller :
		(
		stateRollerInit,
		stateRollerOpening,
		stateRollerOpened,
		stateRollerClosing,
		stateRollerClosed
		);
	StateCentering :
		(
		stateCenteringInit,
		stateCenteringMovingForward,
		stateCenteringForward,
		stateCenteringMovingBack,
		stateCenteringBack
		);
	StateRailing :
		(
		stateRailingInit,
		stateRailingMovingUp,
		stateRailingUp,
		stateRailingMovingDown,
		stateRailingDown
		);
	StateSuckers :
		(
		stateSuckersInit,
		stateSuckersMovingForward,
		stateSuckersForward,
		stateSuckersMovingBack,
		stateSuckersBack
		);
END_TYPE
```

#### Variables.var - Local variables
```iecst
VAR
	diCenteringBack : BOOL;
	diCenteringForward : BOOL;
	diRailingDown : BOOL;
	diRailingUp : BOOL;
	diRollerClosed : BOOL;
	diRollerOpened : BOOL;
	diSuckerLeftBackBack : BOOL;
	diSuckerLeftFrontBack : BOOL;
	diSuckerRightBackBack : BOOL;
	diSuckerRightFrontBack : BOOL;
	doCenetringBack : BOOL;
	doCenetringBrake : BOOL;
	doCenteringBack : BOOL;
	doCenteringForward : BOOL;
	doNoSuck : BOOL;
	DoorLogic_3 : DoorLogic;
	doRailingDown : BOOL;
	doRailingUp : BOOL;
	doRollerBrake : BOOL;
	doRollerClose : BOOL;
	doRollerOpen : BOOL;
	doSuckersBack : BOOL;
	doSuckersForward : BOOL;
	TON_CenteringRequest : TON;
	TON_RailingRequest : TON;
	TON_RollerRequest : TON;
	TON_SuckersRequest : TON;
END_VAR
```

#### Railing.st
```iecst
ACTION Railing:

	IF modeZonePalletization = modeZoneOff THEN
		stateRailing := stateRailingInit;
	END_IF

	CASE stateRailing OF

		stateRailingInit:

			IF diRailingUp AND NOT diRailingDown THEN
				railingUp := TRUE;
				stateRailing := stateRailingUp;
			END_IF

			IF NOT diRailingUp AND diRailingDown THEN
				railingUp := FALSE;
				stateRailing := stateRailingDown;
			END_IF

			//default state
			IF stateRailing = stateRailingInit THEN
				doRailingUp := TRUE;
				doRailingDown := NOT doRailingUp;
			END_IF

		stateRailingMovingUp:

			//set output
			doRailingUp := TRUE;
			doRailingDown := NOT doRailingUp;

			//open check
			IF diRailingUp AND NOT diRailingDown THEN
				stateRailing := stateRailingUp;
			END_IF
			// timer
			TON_RailingRequest(IN := TRUE, PT := T#5s);
			IF TON_RailingRequest.Q THEN
				alarmImagePalletization[8] := TRUE;
				railingUp := FALSE;
				stateRailing := stateRailingDown;
			END_IF

		stateRailingUp:

			// command to go down
			IF NOT railingUp THEN
				TON_RailingRequest(IN := FALSE);
				stateRailing := stateRailingMovingDown;
			END_IF

		stateRailingMovingDown:

			//set output
			doRailingUp := FALSE;
			doRailingDown := NOT doRailingUp;
			// check
			IF NOT diRailingUp AND diRailingDown THEN
				stateRailing := stateRailingDown;
			END_IF
			//timer
			TON_RailingRequest(IN := TRUE, PT := T#5s);
			IF TON_RailingRequest.Q THEN
				alarmImagePalletization[32] := TRUE;
				railingUp := TRUE;
				stateRailing := stateRailingUp;
			END_IF

		stateRailingDown:

			// command to go ip
			IF railingUp THEN
				TON_RailingRequest(IN := FALSE);
				stateRailing := stateRailingMovingUp;
			END_IF
	END_CASE

	//alarms
	IF stateRailing = stateRailingInit THEN
		alarmImagePalletization[33] := TRUE;
	ELSE
		alarmImagePalletization[33] := FALSE;
	END_IF

	//edge alarms
	IF acknowledgeImagePalletization[8] THEN
		alarmImagePalletization[8] := FALSE;
	END_IF
	IF acknowledgeImagePalletization[32] THEN
		alarmImagePalletization[32] := FALSE;
	END_IF

END_ACTION
```

#### Suckers.st
```iecst
ACTION Suckers:

	IF modeZonePalletization = modeZoneOff THEN
		stateSuckers := stateSuckersInit;
	END_IF

	CASE stateSuckers OF

		stateSuckersInit:

			IF diSuckerLeftFrontBack AND diSuckerLeftBackBack AND diSuckerRightFrontBack AND diSuckerRightBackBack THEN
				suckersForward := FALSE;
				stateSuckers := stateSuckersBack;
			END_IF

			IF NOT diSuckerLeftFrontBack AND NOT diSuckerLeftBackBack AND NOT diSuckerRightFrontBack AND NOT diSuckerRightBackBack THEN
				suckersForward := TRUE;
				stateSuckers := stateSuckersForward;
			END_IF

			//default state
			IF stateSuckers = stateSuckersInit THEN
				doSuckersForward := FALSE;
				doSuckersBack := NOT doSuckersForward;
			END_IF

		stateSuckersMovingBack:

			//set output
			doSuckersForward := FALSE;
			doSuckersBack := NOT doSuckersForward;

			// check
			IF diSuckerLeftFrontBack AND diSuckerLeftBackBack AND diSuckerRightFrontBack AND diSuckerRightBackBack THEN
//				suckersForward := FALSE;
				stateSuckers := stateSuckersBack;
			END_IF

			// timer
			TON_SuckersRequest(IN := TRUE, PT := T#5s);
			IF TON_SuckersRequest.Q THEN
				alarmImagePalletization[36] := TRUE;
				suckersForward := TRUE;
				stateSuckers := stateSuckersForward;
			END_IF

		stateSuckersBack:

			// command to go down
			IF suckersForward THEN
				TON_SuckersRequest(IN := FALSE);
				stateSuckers := stateSuckersMovingForward;
			END_IF

		stateSuckersMovingForward:

			//set output
			doSuckersForward := TRUE;
			doSuckersBack := NOT doSuckersForward;

			// check
			IF NOT diSuckerLeftFrontBack AND NOT diSuckerLeftBackBack AND NOT diSuckerRightFrontBack AND NOT diSuckerRightBackBack THEN
//				suckersForward := TRUE;
				stateSuckers := stateSuckersForward;
			END_IF

			//timer
			TON_SuckersRequest(IN := TRUE, PT := T#5s);
			IF TON_SuckersRequest.Q THEN
				alarmImagePalletization[35] := TRUE;
				suckersForward := FALSE;
				stateSuckers := stateSuckersBack;
			END_IF

		stateSuckersForward:

			// command to go ip
			IF NOT suckersForward THEN
				TON_SuckersRequest(IN := FALSE);
				stateSuckers := stateSuckersMovingBack;
			END_IF
	END_CASE

	doNoSuck := NOT doSuck;

	//alarms
	IF stateSuckers = stateSuckersInit THEN
		alarmImagePalletization[34] := TRUE;
	ELSE
		alarmImagePalletization[34] := FALSE;
	END_IF

	//edge alarms
	IF acknowledgeImagePalletization[35] THEN
		alarmImagePalletization[35] := FALSE;
	END_IF
	IF acknowledgeImagePalletization[36] THEN
		alarmImagePalletization[36] := FALSE;
	END_IF

END_ACTION
```

#### Centering.st
```iecst
ACTION Centering:

	IF modeZonePalletization = modeZoneOff THEN
		stateCentering := stateCenteringInit;
	END_IF

	CASE stateCentering OF

		stateCenteringInit:

			IF diCenteringBack THEN
				centeringForward := FALSE;
				stateCentering := stateCenteringBack;
			END_IF

			IF NOT diCenteringBack THEN
				centeringForward := TRUE;
				stateCentering := stateCenteringForward;
			END_IF

			//default state
			IF stateCentering = stateCenteringInit THEN
				doCenteringForward := FALSE;
				doCenetringBack := FALSE;
			END_IF

		stateCenteringMovingBack:

			//set outputs
			doCenteringForward := FALSE;
			doCenteringBack := TRUE;

			// check
			IF diCenteringBack THEN
//				centeringForward := FALSE;
				stateCentering := stateCenteringBack;
			END_IF

			// timer
			TON_CenteringRequest(IN := TRUE, PT := T#6s);
			IF TON_CenteringRequest.Q THEN
				alarmImagePalletization[38] := TRUE;
				centeringForward := TRUE;
				stateCentering := stateCenteringForward;
			END_IF

		stateCenteringBack:

			//set outputs
			doCenteringForward := FALSE;
			doCenteringBack := FALSE;

			// command to go down
			IF centeringForward THEN
				TON_CenteringRequest(IN := FALSE);
				stateCentering := stateCenteringMovingForward;
			END_IF

		stateCenteringMovingForward:

			//set outputs
			doCenteringForward := TRUE;
			doCenteringBack := FALSE;

			//timer
			TON_CenteringRequest(IN := TRUE, PT := T#2s);
			IF TON_CenteringRequest.Q OR diCenteringForward THEN
//				centeringForward := TRUE;
				stateCentering := stateCenteringForward;
			END_IF

		stateCenteringForward:

			//set outputs
			doCenteringForward := FALSE;
			doCenteringBack := FALSE;

			// command to go up
			IF NOT centeringForward THEN
				TON_CenteringRequest(IN := FALSE);
				stateCentering := stateCenteringMovingBack;
			END_IF
	END_CASE

	// brake control
	doCenetringBrake := doCenteringForward OR doCenteringBack;

	//alarms
	IF stateCentering = stateCenteringInit THEN
		alarmImagePalletization[37] := TRUE;
	ELSE
		alarmImagePalletization[37] := FALSE;
	END_IF

	//edge alarms
	IF acknowledgeImagePalletization[38] THEN
		alarmImagePalletization[38] := FALSE;
	END_IF

END_ACTION
```

#### Roller.st
```iecst
ACTION Roller:

	IF modeZonePalletization = modeZoneOff THEN
		stateRoller := stateRollerInit;
	END_IF

	CASE stateRoller OF

		stateRollerInit:

			IF diRollerOpened AND NOT diRollerClosed THEN
				stateRoller := stateRollerOpened;
			END_IF

			IF NOT diRollerOpened AND diRollerClosed  THEN
				stateRoller := stateRollerClosed;
			END_IF

			//default state
			IF stateRoller = stateRollerInit THEN
				IF cmdRollerOpen THEN
					TON_RollerRequest(IN := FALSE);
					stateRoller := stateRollerOpening;
				END_IF

				IF cmdRollerClose THEN
					TON_RollerRequest(IN := FALSE);
					stateRoller := stateRollerClosing;
				END_IF
			END_IF

		stateRollerOpening:

			//set output
			doRollerOpen := TRUE;

			// check
			IF diRollerOpened OR NOT cmdRollerOpen THEN
				StopMovement;
			END_IF

			// timer
			TON_RollerRequest(IN := TRUE, PT := T#6s);
			IF TON_RollerRequest.Q THEN
				alarmImagePalletization[40] := TRUE;
				StopMovement;
			END_IF

			IF stateSuckers <> stateSuckersBack THEN
				alarmImagePalletization[54] := TRUE;
				StopMovement;
			END_IF

		stateRollerOpened:

			IF cmdRollerClose THEN
				TON_RollerRequest(IN := FALSE);
				stateRoller := stateRollerClosing;
			END_IF
			cmdRollerOpen := FALSE;

		stateRollerClosing:

			//set output
			doRollerClose := TRUE;
			//position reached?
			IF diRollerClosed OR NOT cmdRollerClose THEN
				StopMovement;
			END_IF

			// timer
			TON_RollerRequest(IN := TRUE, PT := T#6s);
			IF TON_RollerRequest.Q THEN
				alarmImagePalletization[41] := TRUE;
				StopMovement;
			END_IF

		stateRollerClosed:

			IF cmdRollerOpen THEN
				TON_RollerRequest(IN := FALSE);
				stateRoller := stateRollerOpening;
			END_IF
			cmdRollerClose := FALSE;
	END_CASE

	// brake control
	doRollerBrake := doRollerOpen OR doRollerClose;

	// alarms
	IF acknowledgeImagePalletization[40] THEN
		alarmImagePalletization[40] := FALSE;
	END_IF
	IF acknowledgeImagePalletization[41] THEN
		alarmImagePalletization[41] := FALSE;
	END_IF
	IF acknowledgeImagePalletization[54] THEN
		alarmImagePalletization[54] := FALSE;
	END_IF

END_ACTION

ACTION StopMovement:
	cmdRollerClose := FALSE;
	cmdRollerOpen := FALSE;
	doRollerClose := doRollerOpen :=  FALSE;
	stateRoller := stateRollerInit;
END_ACTION
```

### Program Logical/plc/palletization/robot/robot (IEC) - robot control

#### Types.typ
```iecst
TYPE
	C5GMap_In_typ : 	STRUCT
		NoAlarm : BOOL;
		DriveOnStatus : BOOL;
		Start_NoHoldPrgMove : BOOL;
		Remote : BOOL;
		TeachEnabled : BOOL;
		U1 : BOOL;
		U2 : BOOL;
		U3 : BOOL;
		U4 : BOOL;
		NoLatchAlarmActive : BOOL;
		SafetySpeedActive : BOOL;
		ProgrammingMode : BOOL;
		Reserved : BOOL;
		Local_Remote : BOOL;
		SystemReady : BOOL;
		HeartBit : BOOL;
	END_STRUCT;
	C5GMap_Out_typ : 	STRUCT
		DriveOn : BOOL;
		NoDriveOff : BOOL;
		Start : BOOL;
		NoHold : BOOL;
		U1 : BOOL;
		U2 : BOOL;
		U3 : BOOL;
		U4 : BOOL;
		CancelAlarm : BOOL;
		SafetySpeed : BOOL;
	END_STRUCT;
	C5GMap_DATA_typ : 	STRUCT
		IN : C5GMap_In_typ;
		OUT : C5GMap_Out_typ;
	END_STRUCT;
	C5GMap_RAW_typ : 	STRUCT
		IN : ARRAY[0..IN_SIZE]OF UDINT;
		OUT : ARRAY[0..OUT_SIZE]OF UDINT;
	END_STRUCT;
	C5GMap_typ : 	STRUCT
		ModuleOk : BOOL;
		Data : C5GMap_DATA_typ;
		Raw : C5GMap_RAW_typ;
	END_STRUCT;
END_TYPE
```

#### Variables.var
```iecst
VAR
	Comau_0 : Comau;
	dActualRecipe : REFERENCE TO Recipe;
	diSeparatorPresent : BOOL;
	dRecipes : REFERENCE TO Recipes;
	ModuleOk : BOOL;
	MTBasicsPWM_0 : MTBasicsPWM;
	MTBasicsPWM_1 : MTBasicsPWM;
	robotDoorEdmError : BOOL;
	robotEdmError : BOOL;
	TON_Robot : TON;
	tmpBOOL : BOOL;
END_VAR
```

#### Main.st
```iecst
PROGRAM _INIT

	Comau_0.NoDriveOff := TRUE;

END_PROGRAM

PROGRAM _CYCLIC

	IF adrRecipes = 0 THEN
		RETURN;
	END_IF

	dRecipes ACCESS adrRecipes;
	IF dRecipes.actualRecipeIndex < 0 OR dRecipes.actualRecipeIndex > 9 THEN
		RETURN;
	END_IF

	dActualRecipe ACCESS ADR(dRecipes.recipe[dRecipes.actualRecipeIndex]);

	Comau_0.ProductType := INT_TO_USINT(dRecipes.actualRecipeIndex+1);

	//drive on
	MTBasicsPWM_1(Enable :=  Comau_0.NoAlarm AND NOT Comau_0.DriveOnStatus, Period := 1, DutyCycle := 50);
	Comau_0.DriveOn := MTBasicsPWM_1.Out;

	IF statePalletP14 <> palletPresent THEN
		palletComplete := FALSE;
	END_IF

	CASE modeZonePalletization OF

		modeZoneOff:

			//stateRobotAuto := stateRobotAutoInit;

		modeZoneManual:

			IF modeZonePalletizationOld <> modeZoneManual THEN
				Comau_0.MakeMove := FALSE;
//				doSuck := FALSE;
			END_IF

			Comau_0.NoHold := Comau_0.ProgrammingMode;

			IF Comau_0.ProgrammingMode THEN
				stateRobotAuto := stateRobotAutoInit;
			END_IF

		modeZoneAuto:

			Comau_0.NoHold := TRUE;

			CASE stateRobotAuto OF

				stateRobotAutoInit:

					stateRobotAuto := stateRobotAutoGoHome;

				stateRobotAutoGoHome:

					IF Comau_0.IsItSafeToGoHome THEN
						stateRobotAuto := stateRobotAutoGoHome2;
					ELSE
						alarmImagePalletization[49] := TRUE;
					END_IF

				stateRobotAutoGoHome2:

					Comau_0.MoveType := moveTypeGoHome;
					Comau_0.MakeMove := TRUE;

					IF Comau_0.MoveDone THEN
						stateRobotAuto := stateRobotAutoPrepareHead;
					END_IF

				stateRobotAutoPrepareHead:

					IF nbOfTraysInRobotHead > 0 THEN

						suckersForward := TRUE;

						IF stateSuckers = stateSuckersForward THEN
							stateRobotAuto := stateRobotAutoPreGoToTable;
						END_IF

						stateRobotAuto := stateRobotAutoPreGoToTable;

					ELSE
						suckersForward := TRUE;
						railingUp := TRUE;
						centeringForward := FALSE;
						cmdRollerClose := TRUE;
						doSuck := FALSE;

						IF (suckersForward = TRUE) AND (railingUp = TRUE) AND (centeringForward = FALSE) AND (doSuck = FALSE) THEN
							stateRobotAuto := stateRobotAutoPreGoToTable;
						END_IF
					END_IF

				stateRobotAutoPreGoToTable:

					Comau_0.MoveType := moveTypeGoToTable;
					Comau_0.MakeMove := TRUE;

					IF Comau_0.MoveDone THEN
						stateRobotAuto := stateRobotAutoGoingToTable;
					END_IF

				stateRobotAutoGoingToTable:
					IF (stateSuckers = stateSuckersForward AND stateRailing = stateRailingUp AND stateCentering = stateCenteringBack AND stateRoller = stateRollerClosed) OR cpuIsSimulated THEN
						stateRobotAuto := stateRobotAutoGoToTable;
					END_IF

				stateRobotAutoGoToTable:

					Comau_0.MoveType := moveTypeEndGoToTable;
					Comau_0.MakeMove := TRUE;

					IF Comau_0.MoveDone THEN
						stateRobotAuto := stateRobotAutoWaitForBottles;
					END_IF

				stateRobotAutoWaitForBottles:

					//head full?
					IF nbOfTraysInRobotHead > 0 THEN

						robotData.layer := nbOfLayersOnPallet;
						robotData.placeFirstHalf := nbOfTraysInHalfLayer = 0;

						IF nbOfLayersOnPallet = 0 THEN
							robotData.placeSeparator := dActualRecipe.interlayerSheetBottom;
						ELSE
							robotData.placeSeparator := TRUE;
						END_IF

						IF NOT robotData.placeFirstHalf THEN
							robotData.placeSeparator := FALSE;
						END_IF

						IF nbOfLayersOnPallet = dActualRecipe.nbOfLayers - 1 THEN
							robotData.placeSeparatorAbove := dActualRecipe.interlayerSheetTop;
						ELSE
							robotData.placeSeparatorAbove := FALSE;
						END_IF

						IF robotData.placeFirstHalf THEN
							robotData.placeSeparatorAbove := FALSE;
						END_IF

						Comau_0.NbOfLayers := INT_TO_USINT(robotData.layer);

						stateRobotAuto := stateRobotAutoRailingDown;
					END_IF

				stateRobotAutoRailingDown:

					railingUp := FALSE;

					IF stateRailing = stateRailingDown OR cpuIsSimulated THEN
						stateRobotAuto := stateRobotAutoCenteringForward;
					END_IF

				stateRobotAutoCenteringForward:

					centeringForward := TRUE;

					IF stateCentering = stateCenteringForward OR cpuIsSimulated THEN
						stateRobotAuto := stateRobotAutoSwitch1;
					END_IF

				stateRobotAutoSwitch1:

					IF robotData.placeFirstHalf AND robotData.placeSeparator THEN
						stateRobotAuto := stateRobotAutoSeparator;
					ELSE
						stateRobotAuto := stateRobotAutoHideSuckers;
					END_IF

				stateRobotAutoSeparator:

					Comau_0.MoveType := moveTypeGoForSeparator;
					Comau_0.MakeMove := TRUE;

					IF Comau_0.MoveDone THEN
						stateRobotAuto := stateRobotAutoSeparator2;
					END_IF

				stateRobotAutoSeparator2:

					doSuck := TRUE;

					TON_Robot(IN := TRUE, PT := T#0.2s);
					IF TON_Robot.Q THEN
						stateRobotAuto := stateRobotAutoSeparator3;
					END_IF

				stateRobotAutoSeparator3:

					Comau_0.MoveType := moveTypeVerticalOffset2;
					Comau_0.MakeMove := TRUE;

					IF Comau_0.MoveDone THEN
						stateRobotAuto := stateRobotAutoSeparator4;
					END_IF

				stateRobotAutoSeparator4:

					IF diSeparatorPresent THEN
						stateRobotAuto := stateRobotAutoSeparator5;
					ELSE
						alarmImagePalletization[52] := TRUE;
						stateRobotAuto := stateRobotAutoSeparator;
					END_IF

				stateRobotAutoSeparator5:

					IF statePalletP14 = palletPresent AND NOT palletComplete THEN
						stateRobotAuto := stateRobotAutoSeparator6;
					END_IF

				stateRobotAutoSeparator6:

					Comau_0.MoveType := moveTypePutSeparatorOnPallet;
					Comau_0.MakeMove := TRUE;

					IF Comau_0.MoveDone THEN
						doSuck := FALSE;
						stateRobotAuto := stateRobotAutoHideSuckers;
					END_IF

				stateRobotAutoHideSuckers:

					Comau_0.MoveType := moveTypeVerticalOffset;
					Comau_0.MakeMove := TRUE;

					IF Comau_0.MoveDone THEN
						IF robotData.placeSeparatorAbove AND Comau_0.NbOfLayers = INT_TO_USINT(robotData.layer) + 1 THEN
							palletComplete := TRUE;
							stateRobotAuto := stateRobotAutoPrepareHead;
						ELSE
							stateRobotAuto := stateRobotAutoHideSuckers2;
						END_IF
					END_IF

				stateRobotAutoHideSuckers2:

					suckersForward := FALSE;

					IF stateSuckers = stateSuckersBack OR cpuIsSimulated THEN
						stateRobotAuto := stateRobotAutoWaitForPallet;
					END_IF

				stateRobotAutoWaitForPallet:

					IF statePalletP14 = palletPresent AND NOT palletComplete THEN
						IF robotData.placeFirstHalf THEN
							stateRobotAuto := stateRobotAutoPlaceFirstHalf;
						ELSE
							stateRobotAuto := stateRobotAutoPlaceSecondHalf;
						END_IF
					END_IF

				stateRobotAutoPlaceFirstHalf:

					Comau_0.MoveType := moveTypePlaceFirstHalf;
					Comau_0.MakeMove := TRUE;

					IF Comau_0.MoveDone THEN
						stateRobotAuto := stateRobotAutoPlaceFirstHalf2;
					END_IF

				stateRobotAutoPlaceFirstHalf2:

					cmdRollerOpen := TRUE;

					IF stateRoller = stateRollerOpened OR cpuIsSimulated THEN
						stateRobotAuto := stateRobotAutoPlaceFirstHalf3;
					END_IF

				stateRobotAutoPlaceFirstHalf3:

					railingUp := TRUE;
					centeringForward := FALSE;

					IF (stateRailing = stateRailingUp AND stateCentering = stateCenteringBack) OR cpuIsSimulated THEN
						stateRobotAuto := stateRobotAutoPlaceFirstHalf4;
					END_IF

				stateRobotAutoPlaceFirstHalf4:

					Comau_0.MoveType := moveTypeVerticalOffset2;
					Comau_0.MakeMove := TRUE;

					IF Comau_0.MoveDone THEN
						counterTraysOnPallet := counterTraysInRobotHead;

						stateRobotAuto := stateRobotAutoPrepareHead;
					END_IF

				stateRobotAutoPlaceSecondHalf:

					Comau_0.MoveType := moveTypePlaceSecondHalf;
					Comau_0.MakeMove := TRUE;

					IF Comau_0.MoveDone THEN
						stateRobotAuto := stateRobotAutoPlaceSecondHalf2;
					END_IF

				stateRobotAutoPlaceSecondHalf2:

					railingUp := TRUE;

					IF stateRailing = stateRailingUp OR cpuIsSimulated THEN
						stateRobotAuto := stateRobotAutoPlaceSecondHalf3;
					END_IF

				stateRobotAutoPlaceSecondHalf3:

					Comau_0.MoveType := moveTypeRelativeHorizontalOffset;
					Comau_0.MakeMove := TRUE;

					IF Comau_0.MoveDone THEN
						stateRobotAuto := stateRobotAutoPlaceSecondHalf4;
					END_IF

				stateRobotAutoPlaceSecondHalf4:

					cmdRollerOpen := TRUE;

					IF stateRoller = stateRollerOpened OR cpuIsSimulated THEN
						stateRobotAuto := stateRobotAutoPlaceSecondHalf5;
					END_IF

				stateRobotAutoPlaceSecondHalf5:

					centeringForward := FALSE;

					IF stateCentering = stateCenteringBack OR cpuIsSimulated THEN
						stateRobotAuto := stateRobotAutoPlaceSecondHalf6;
					END_IF

				stateRobotAutoPlaceSecondHalf6:

					Comau_0.MoveType := moveTypeVerticalOffset2;
					Comau_0.MakeMove := TRUE;

					IF Comau_0.MoveDone THEN

						counterTraysOnPallet := counterTraysInRobotHead;

						IF robotData.placeSeparatorAbove THEN
							stateRobotAuto := stateRobotAutoSeparatorAbove;
						ELSE
							IF counterTraysInRobotHead MOD nbOfTraysInCompletePallet = 0 THEN
								counterTraysInRobotHead := 0;
								palletComplete := TRUE;
							END_IF
							stateRobotAuto := stateRobotAutoPrepareHead;
						END_IF

					END_IF

				stateRobotAutoSeparatorAbove:

					Comau_0.NbOfLayers := INT_TO_USINT(robotData.layer) + 1;

					suckersForward := TRUE;
					railingUp := TRUE;
					centeringForward := FALSE;
					cmdRollerClose := TRUE;
					doSuck := FALSE;

					IF stateSuckers = stateSuckersForward AND stateRailing = stateRailingUp AND stateCentering = stateCenteringBack AND stateRoller = stateRollerClosed THEN
						stateRobotAuto := stateRobotAutoSeparator;
					END_IF

			END_CASE

			IF (pusherDrive.actualPositionIndex > 3 OR pusherDrive.requestedPositionIndex > 3) AND stateRobotAuto <> stateRobotAutoWaitForBottles THEN
				alarmImagePalletization[53] := TRUE;
			END_IF

	END_CASE

	IF Comau_0.MoveDone THEN
		Comau_0.MakeMove := FALSE;
	END_IF

	IF TON_Robot.Q THEN
		TON_Robot(IN := FALSE);
	END_IF

	Comau_0();

	IF cpuIsSimulated THEN
		tmpBOOL := TRUE;
		memcpy(ADR(Comau_0.MoveDone),ADR(tmpBOOL), SIZEOF(tmpBOOL));
		memcpy(ADR(Comau_0.IsItSafeToGoHome),ADR(tmpBOOL), SIZEOF(tmpBOOL));
	END_IF

	//alarms
	alarmImagePalletization[50] := NOT ModuleOk;
	alarmImagePalletization[45] := robotEdmError;
	alarmImagePalletization[46] := robotDoorEdmError;
	alarmImagePalletization[47] := NOT Comau_0.Remote;
	alarmImagePalletization[48] := NOT Comau_0.NoAlarm;

	IF Comau_0.Error THEN
		alarmImagePalletization[51] := TRUE;
	END_IF

	IF Comau_0.ErrorHoldPressed THEN
		alarmImagePalletization[56] := TRUE;
	END_IF

	MTBasicsPWM_0(Enable :=  alarmImagePalletization[48] AND NOT acknowledgeImagePalletization[48], Period := 1, DutyCycle := 50);
	Comau_0.CancelAlarm := MTBasicsPWM_0.Out;

	//edge alarms
	IF acknowledgeImagePalletization[49] THEN
		alarmImagePalletization[49] := FALSE;
	END_IF

	IF acknowledgeImagePalletization[51] THEN
		alarmImagePalletization[51] := FALSE;
	END_IF

	IF acknowledgeImagePalletization[52] THEN
		alarmImagePalletization[52] := FALSE;
	END_IF
	IF acknowledgeImagePalletization[53] THEN
		alarmImagePalletization[53] := FALSE;
	END_IF

	IF acknowledgeImagePalletization[56] THEN
		alarmImagePalletization[56] := FALSE;
	END_IF

	IF testAtAtrima THEN
		alarmImagePalletization[47] := FALSE;
		alarmImagePalletization[48] := FALSE;
		alarmImagePalletization[49] := FALSE;
	END_IF

END_PROGRAM
```

### Program Logical/plc/palletization/pallet_conveyors/pallet_conveyors (IEC) - pallet conveyors control

#### Main.st - Cyclic code
```iecst
PROGRAM _INIT
	(* Insert code here *)

END_PROGRAM

PROGRAM _CYCLIC

	CASE modePalletization OF

		modePalletizationNotReadyToStart: //the automat is not ready to start

			(***************************************************************************)
			(* 								Pallet Status							   *)
			(***************************************************************************)
			CopyToArray;

		modePalletizationManual:

			IF modePalletizationOld <> modePalletizationManual THEN
				cmdMovePalletP12 := FALSE;
				cmdMovePalletP13 := FALSE;
				cmdMovePalletP14 := FALSE;
			END_IF

			(***************************************************************************)
			(* 								Pallet Status							   *)
			(***************************************************************************)
			FOR i:=12 TO 22 DO
				IF (PalletStatus[i] <> PalletStatus_old[i]) THEN
					IF ((PalletStatus[i]) = 3) THEN
						PalletStatus[i] := 0;
					END_IF;
					PalletStatus_old[i] := PalletStatus[i];
				END_IF;
			END_FOR;
			CopyFromArray;

		modePalletizationAuto:

			IF statePalletP12 <> palletNotPresent AND statePalletP13 = palletNotPresent THEN
				cmdMovePalletP12 := TRUE;
			END_IF

			IF statePalletP13 <> palletNotPresent AND statePalletP14 = palletNotPresent THEN
				cmdMovePalletP13 := TRUE;
			END_IF

			IF statePalletP14 <> palletNotPresent AND statePalletP15 = palletNotPresent THEN
				cmdMovePalletP14 := TRUE;
			END_IF

			CopyToArray;
	END_CASE

	//conveyors
	ConveyorP12Control;
	ConveyorP13Control;
	ConveyorP14Control;
	ConveyorP15Control;
	ConveyorP16Control;

	alarmImagePalletization[5] := NOT lightCurtainP15;
	alarmImagePalletization[8] := NOT lightCurtainP17;

END_PROGRAM
```

#### Variables.var - Local variables
```iecst
VAR
	acpI_P14 : AcpInoSdc;
	acpI_P15 : AcpInoSdc;
	acpI_P16 : AcpInoSdc;
	cmdMovePalletP12 : BOOL;
	cmdMovePalletP13 : BOOL;
	cmdMovePalletP14 : BOOL;
	cmdMovePalletP15 : BOOL;
	diMotorProtectionP12 : BOOL;
	diMotorProtectionP13 : BOOL;
	diPalletSlowDownP14 : BOOL;
	diPalletStopP13 : BOOL;
	diPalletStopP14 : BOOL;
	diPalletStopP15 : BOOL;
	diPalletStopP16 : BOOL;
	doConveyorP12 : BOOL; (*starts conveyor P12*)
	doConveyorP13 : BOOL;
	lightCurtainP15 : BOOL;
	lightCurtainP17 : BOOL;
	palletStopP13old : BOOL;
	palletStopP14old : BOOL;
	palletStopP15old : BOOL;
	palletStopP16old : BOOL;
	TON_ConveyorP12 : TON;
	TON_ConveyorP13 : TON;
	TON_ConveyorP14 : TON;
	TON_ConveyorP15 : TON;
	TON_PalletStopP13 : TON;
	TON_PalletStopP14 : TON;
	TON_PalletStopP15 : TON;
	TON_PalletStopP16 : TON;
	diPalletStopP17 : BOOL;
	TON_PalletStopP17 : TON;
	palletStopP17old : BOOL;
	cmdMovePalletP16 : BOOL;
	TON_ConveyorP16 : TON;
	acpI_P17 : AcpInoSdc;
	cmdMovePalletP17 : BOOL;
	i : INT;
END_VAR
```

#### VisuCorrection.st
```iecst
ACTION CopyToArray:

	PalletStatus[12] := statePalletP12;
	PalletStatus[13] := statePalletP13;
	PalletStatus[14] := statePalletP14;
	PalletStatus[15] := statePalletP15;
	PalletStatus[16] := statePalletP16;
	PalletStatus[17] := statePalletP17;
END_ACTION

ACTION CopyFromArray:

	statePalletP12 := PalletStatus[12];
	statePalletP13 := PalletStatus[13];
	statePalletP14 := PalletStatus[14];
	statePalletP15 := PalletStatus[15];
	statePalletP16 := PalletStatus[16];
	statePalletP17 := PalletStatus[17];

END_ACTION
```

#### conveyorP12Control.st
```iecst
ACTION ConveyorP12Control:

	TON_PalletStopP13(IN := diPalletStopP13, PT := T#200ms);

	CASE statePalletP12 OF

		palletNotPresent:

			doConveyorP12 := cmdMovePalletP12 AND (statePalletP13 = palletNotPresent OR diReset);

		palletPresent:

			doConveyorP12 := FALSE;

			IF cmdMovePalletP12 AND (statePalletP13 = palletNotPresent OR diReset) THEN
				TON_ConveyorP12(IN := FALSE);
				statePalletP12 := palletMoving;
			END_IF

		palletMoving:

			//sensor reached?
			IF TON_PalletStopP13.Q AND NOT diReset THEN
				statePalletP13 := palletPresent;
				statePalletP12 := palletNotPresent;
				cmdMovePalletP12 := FALSE;
			END_IF

			//timeout?
			IF modePalletization = modePalletizationAuto THEN
				TON_ConveyorP12(IN := TRUE, PT := T#12s);
				IF TON_ConveyorP12.Q THEN
					alarmImagePalletization[0] := TRUE;
					cmdMovePalletP12 := FALSE;
				END_IF
			ELSE
				TON_ConveyorP12(IN := FALSE);
			END_IF

			doConveyorP12 := cmdMovePalletP12;

	END_CASE

	IF EDGEPOS(TON_PalletStopP13.Q) AND statePalletP12 <> palletMoving THEN
		alarmImagePalletization[9] := TRUE;
	END_IF

	alarmImagePalletization[12] := NOT diMotorProtectionP12;

	//edge alarms
	IF acknowledgeImagePalletization[0] THEN
		alarmImagePalletization[0] := FALSE;
	END_IF

	IF acknowledgeImagePalletization[9] THEN
		alarmImagePalletization[9] := FALSE;
	END_IF

END_ACTION
```

#### conveyorP13Control.st
```iecst
ACTION ConveyorP13Control:

	TON_PalletStopP14(IN := diPalletStopP14, PT := T#200ms);

	CASE statePalletP13 OF

		palletNotPresent:

			doConveyorP13 := (cmdMovePalletP13 AND (statePalletP14 = palletNotPresent OR diReset)) OR cmdMovePalletP12;

		palletPresent:

			doConveyorP13 := FALSE;

			IF cmdMovePalletP13 AND (statePalletP14 = palletNotPresent OR diReset) THEN
				TON_ConveyorP13(IN := FALSE);
				statePalletP13 := palletMoving;
			END_IF

		palletMoving:

			//slow down sensor?
			IF diPalletSlowDownP14 THEN
				acpI_P14.speed := 200;
			END_IF

			//sensor reached?
			IF TON_PalletStopP14.Q AND NOT diReset THEN
				statePalletP14 := palletPresent;
				statePalletP13 := palletNotPresent;
				cmdMovePalletP13 := FALSE;
			END_IF

			//timeout?
			IF modePalletization = modePalletizationAuto THEN
				TON_ConveyorP13(IN := TRUE, PT := T#12s);
				IF TON_ConveyorP13.Q THEN
					alarmImagePalletization[2] := TRUE;
					cmdMovePalletP13 := FALSE;
				END_IF
			ELSE
				TON_ConveyorP13(IN := FALSE);
			END_IF

			doConveyorP13 := cmdMovePalletP13;

	END_CASE

	IF EDGEPOS(TON_PalletStopP14.Q) AND statePalletP13 <> palletMoving THEN
		alarmImagePalletization[10] := TRUE;
	END_IF

	alarmImagePalletization[13] := NOT diMotorProtectionP13;

	//edge alarms
	IF acknowledgeImagePalletization[2] THEN
		alarmImagePalletization[2] := FALSE;
	END_IF

	IF acknowledgeImagePalletization[10] THEN
		alarmImagePalletization[10] := FALSE;
	END_IF

END_ACTION
```

#### conveyorP14Control.st
```iecst
ACTION ConveyorP14Control:

	TON_PalletStopP15(IN := diPalletStopP15, PT := T#200ms);

	acpI_P14.switchOn := TRUE;
	acpI_P14.speed := 500;

	CASE statePalletP14 OF

		palletNotPresent:

			acpI_P14.stop := NOT (cmdMovePalletP14 AND (statePalletP15 = palletNotPresent OR diReset)) AND NOT cmdMovePalletP13;

		palletPresent:

			acpI_P14.stop := TRUE;

			IF cmdMovePalletP14 AND (statePalletP15 = palletNotPresent OR diReset) THEN
				TON_ConveyorP14(IN := FALSE);
				statePalletP14 := palletMoving;
			END_IF

		palletMoving:

			//sensor reached?
			IF TON_PalletStopP15.Q AND NOT diReset THEN
				statePalletP15 := palletPresent;
				statePalletP14 := palletNotPresent;
				cmdMovePalletP14 := FALSE;
			END_IF

			//timeout?
			IF modePalletization = modePalletizationAuto THEN
				TON_ConveyorP14(IN := TRUE, PT := T#12s);
				IF TON_ConveyorP14.Q THEN
					alarmImagePalletization[7] := TRUE;
					cmdMovePalletP14 := FALSE;
				END_IF
			ELSE
				TON_ConveyorP14(IN := FALSE);
			END_IF

			acpI_P14.stop := NOT cmdMovePalletP14;

	END_CASE

	//control of ACOPOSinverter
	acpI_P14();

	alarmImagePalletization[24] := acpI_P14.error;

	IF EDGEPOS(TON_PalletStopP15.Q) AND statePalletP14 <> palletMoving THEN
		alarmImagePalletization[11] := TRUE;
	END_IF

	//edge alarms
	IF acknowledgeImagePalletization[7] THEN
		alarmImagePalletization[7] := FALSE;
	END_IF

	IF acknowledgeImagePalletization[11] THEN
		alarmImagePalletization[11] := FALSE;
	END_IF

	IF EDGENEG(acknowledgeImagePalletization[24]) THEN
		acpI_P14.reset := TRUE;
	END_IF

END_ACTION
```

#### conveyorP15Control.st
```iecst
ACTION ConveyorP15Control:

	TON_PalletStopP16(IN := diPalletStopP16, PT := T#200ms);

	acpI_P15.switchOn := TRUE;
	acpI_P15.speed := 500;

	CASE statePalletP15 OF

		palletNotPresent:

			acpI_P15.stop := NOT (cmdMovePalletP15 AND (statePalletP16 = palletNotPresent OR diReset)) AND NOT cmdMovePalletP14;

		palletPresent:

			acpI_P15.stop := TRUE;

			IF cmdMovePalletP15 AND (statePalletP16 = palletNotPresent OR diReset) THEN
				TON_ConveyorP15(IN := FALSE);
				statePalletP15 := palletMoving;
			END_IF

		palletMoving:

			//sensor reached?
			IF TON_PalletStopP16.Q AND NOT diReset THEN
				statePalletP16 := palletPresent;
				statePalletP15 := palletNotPresent;
				cmdMovePalletP15 := FALSE;
			END_IF

			//timeout?
			IF modePalletization = modePalletizationAuto THEN
				TON_ConveyorP15(IN := TRUE, PT := T#12s);
				IF TON_ConveyorP15.Q THEN
					alarmImagePalletization[3] := TRUE;
					cmdMovePalletP15 := FALSE;
				END_IF
			ELSE
				TON_ConveyorP15(IN := FALSE);
			END_IF

			acpI_P15.stop := NOT cmdMovePalletP15;

	END_CASE

	//control of ACOPOSinverter
	acpI_P15();

	alarmImagePalletization[25] := acpI_P15.error;

	IF EDGEPOS(TON_PalletStopP16.Q) AND statePalletP15 <> palletMoving THEN
		alarmImagePalletization[1] := TRUE;
	END_IF

	//edge alarms
	IF acknowledgeImagePalletization[3] THEN
		alarmImagePalletization[3] := FALSE;
	END_IF

	IF acknowledgeImagePalletization[1] THEN
		alarmImagePalletization[1] := FALSE;
	END_IF

	IF EDGENEG(acknowledgeImagePalletization[25]) THEN
		acpI_P15.reset := TRUE;
	END_IF

END_ACTION
```

#### conveyorP16Control.st
```iecst
ACTION ConveyorP16Control:

	TON_PalletStopP17(IN := diPalletStopP17, PT := T#200ms);

	acpI_P16.switchOn := TRUE;
	acpI_P16.speed := 500;

	CASE statePalletP16 OF

		palletNotPresent:

			acpI_P16.stop := NOT (cmdMovePalletP16 AND (statePalletP17 = palletNotPresent OR diReset)) AND NOT cmdMovePalletP15;

		palletPresent:

			acpI_P16.stop := TRUE;

			IF cmdMovePalletP16 AND (statePalletP17 = palletNotPresent OR diReset) THEN
				TON_ConveyorP16(IN := FALSE);
				statePalletP16 := palletMoving;
			END_IF

		palletMoving:

			//sensor reached?
			IF TON_PalletStopP17.Q AND NOT diReset THEN
				statePalletP17 := palletPresent;
				statePalletP16 := palletNotPresent;
				cmdMovePalletP16 := FALSE;
			END_IF

			//timeout?
			IF modePalletization = modePalletizationAuto THEN
				TON_ConveyorP16(IN := TRUE, PT := T#12s);
				IF TON_ConveyorP16.Q THEN
					alarmImagePalletization[6] := TRUE;
					cmdMovePalletP16 := FALSE;
				END_IF
			ELSE
				TON_ConveyorP16(IN := FALSE);
			END_IF

			acpI_P16.stop := NOT cmdMovePalletP16;

	END_CASE

	//control of ACOPOSinverter
	acpI_P16();

	alarmImagePalletization[26] := acpI_P16.error;

	IF EDGEPOS(TON_PalletStopP17.Q) AND statePalletP16 <> palletMoving THEN
		alarmImagePalletization[4] := TRUE;
	END_IF

	//edge alarms
	IF acknowledgeImagePalletization[6] THEN
		alarmImagePalletization[6] := FALSE;
	END_IF

	IF acknowledgeImagePalletization[4] THEN
		alarmImagePalletization[4] := FALSE;
	END_IF

	IF EDGENEG(acknowledgeImagePalletization[26]) THEN
		acpI_P16.reset := TRUE;
	END_IF

END_ACTION
```

#### conveyorP17Control.st
```iecst
ACTION ConveyorP17Control:

//	TON_PalletStopP17(IN := diPalletStopP17, PT := T#200ms);

	acpI_P17.switchOn := TRUE;
	acpI_P17.speed := 500;

	CASE statePalletP17 OF

		palletNotPresent:

//			acpI_P16.stop := NOT (cmdMovePalletP16 AND (statePalletP17 = palletNotPresent OR diReset)) AND NOT cmdMovePalletP15;

			acpI_P17.stop := NOT cmdMovePalletP17 AND NOT cmdMovePalletP16;

		palletPresent:

//			acpI_P16.stop := TRUE;
//
//			IF cmdMovePalletP16 AND (statePalletP17 = palletNotPresent OR diReset) THEN
//				TON_ConveyorP16(IN := FALSE);
//				statePalletP16 := palletMoving;
//			END_IF

		palletMoving:

//			//sensor reached?
//			IF TON_PalletStopP17.Q AND NOT diReset THEN
//				statePalletP17 := palletPresent;
//				statePalletP16 := palletNotPresent;
//				cmdMovePalletP16 := FALSE;
//			END_IF
//
//			//timeout?
//			IF modePalletization = modePalletizationAuto THEN
//				TON_ConveyorP16(IN := TRUE, PT := T#12s);
//				IF TON_ConveyorP16.Q THEN
//					alarmImagePalletization[6] := TRUE;
//					cmdMovePalletP16 := FALSE;
//				END_IF
//			ELSE
//				TON_ConveyorP16(IN := FALSE);
//			END_IF
//
//			acpI_P16.stop := NOT cmdMovePalletP16;

	END_CASE

	//control of ACOPOSinverter
	acpI_P17();

	alarmImagePalletization[29] := acpI_P16.error;

//	IF EDGEPOS(TON_PalletStopP17.Q) AND statePalletP17 <> palletMoving THEN
//		alarmImagePalletization[4] := TRUE;
//	END_IF

//	palletStopP17old := TON_PalletStopP17.Q;

	//edge alarms
//	IF acknowledgeImagePalletization[6] THEN
//		alarmImagePalletization[6] := FALSE;
//	END_IF
//
//	IF acknowledgeImagePalletization[4] THEN
//		alarmImagePalletization[4] := FALSE;
//	END_IF

	IF EDGENEG(acknowledgeImagePalletization[29]) THEN
		acpI_P17.reset := TRUE;
	END_IF

END_ACTION
```

#### conveyorP12.st - not listed in the package file held
```iecst
ACTION ConveyorP12:

	CASE statePalletP12 OF

		palletNotPresent:

			doConveyorP12 := cmdMovePalletP12 AND (statePalletP13 = palletNotPresent OR diReset);

		palletPresent:

			IF cmdMovePalletP12 AND (statePalletP13 = palletNotPresent OR diReset) THEN
				statePalletP12 := palletMoving;
			END_IF

			doConveyorP12 := FALSE;

		palletMoving:

			//sensor reached?
			IF TON_PalletStopP13.Q AND cmdMovePalletP12 AND NOT diReset THEN
				statePalletP13 := palletPresent;
				statePalletP12 := palletNotPresent;
				cmdMovePalletP12 := FALSE;
			END_IF

			doConveyorP12 := cmdMovePalletP12;

	END_CASE

END_ACTION
```

#### conveyorP12P13Control.st - not listed in the package file held
```iecst
ACTION ConveyorP12P13Control:

	IF modePalletization = modePalletizationNotReadyToStart THEN
		statePalletP12 := palletNotPresent;
	END_IF

	CASE statePalletP12 OF

		palletNotPresent:

			doConveyorP12 := FALSE;
			doConveyorP13 := FALSE;

			IF cmdMovePalletP12P13 THEN
				IF statePalletP13 = palletPresent AND NOT diReset THEN
					alarmImagePalletization[1] := TRUE;
					cmdMovePalletP12P13 := FALSE;
				ELSE
					TON_ConveyorP12P13(IN := FALSE);
					statePalletP12 := palletMoving;
				END_IF
			END_IF

			IF diPalletStopP13 THEN
				alarmImagePalletization[9] := TRUE;
			END_IF

		palletPresent:

			doConveyorP12 := FALSE;
			doConveyorP13 := FALSE;

			IF cmdMovePalletP12P13 THEN
				IF statePalletP13 = palletPresent AND NOT diReset THEN
					alarmImagePalletization[1] := TRUE;
//					statePalletP12 := stateConveyorStop;
				ELSE
					TON_ConveyorP12P13(IN := FALSE);
					statePalletP12 := palletMoving;
				END_IF
			END_IF

		palletMoving:

			IF cmdMovePalletP12P13 THEN
				doConveyorP12 := TRUE;
				doConveyorP13 := TRUE;
			ELSE
				statePalletP12 := palletNotPresent;
			END_IF

			//sensor reached?
			IF diPalletStopP13 AND NOT diReset THEN
				statePalletP13 := palletPresent;
				statePalletP12 := palletNotPresent;
			END_IF

			//timeout?
			TON_ConveyorP12P13(IN := TRUE, PT := T#12s);
			IF TON_ConveyorP12P13.Q AND NOT diReset THEN
				alarmImagePalletization[0] := TRUE;
				cmdMovePalletP12P13 := FALSE;
			END_IF

	END_CASE

	alarmImagePalletization[12] := NOT diMotorProtectionP12;

	//edge alarms
	IF acknowledgeImagePalletization[0] THEN
		alarmImagePalletization[0] := FALSE;
	END_IF
	IF acknowledgeImagePalletization[1] THEN
		alarmImagePalletization[1] := FALSE;
	END_IF
	IF acknowledgeImagePalletization[9] THEN
		alarmImagePalletization[9] := FALSE;
	END_IF

END_ACTION
```

#### conveyorP13.st - not listed in the package file held
```iecst
ACTION ConveyorP13:

	CASE statePalletP13 OF

		palletNotPresent:

			doConveyorP13 := (cmdMovePalletP13 AND (statePalletP14 = palletNotPresent OR diReset)) OR cmdMovePalletP12;

		palletPresent:

			IF cmdMovePalletP13 AND (statePalletP14 = palletNotPresent OR diReset) THEN
				statePalletP13 := palletMoving;
			END_IF

			doConveyorP13 := FALSE;

		palletMoving:

			//sensor reached?
			IF TON_PalletStopP14.Q AND cmdMovePalletP13 AND NOT diReset THEN
				statePalletP14 := palletPresent;
				statePalletP13 := palletNotPresent;
				cmdMovePalletP13 := FALSE;
			END_IF

			doConveyorP13 := cmdMovePalletP13;

	END_CASE

END_ACTION
```
